TEXTLIST S3_Alarms
  0 = 'S3 0 Row 1 Failed To Advance.. Check Qxxx.x Default' | German: 'S3 0 Row 1 Failed To Advance.. Check Qxxx.x German' | French: 'S3 0 Row 1 Failed To Advance.. Check Qxxx.x French'
  1 = 'S3 1 Row 1 Failed To Return.. Check Qxxx.x Default' | German: 'S3 1 Row 1 Failed To Return.. Check Qxxx.x German' | French: 'S3 1 Row 1 Failed To Return.. Check Qxxx.x French'
  2 = 'S3 2 Row 1 Lost Advance Position... Check Ixxx.x Default' | German: 'S3 2 Row 1 Lost Advance Position... Check Ixxx.x German' | French: 'S3 2 Row 1 Lost Advance Position... Check Ixxx.x French'
  3 = 'S3 3 Row 1 Lost Return Position... Check Ixxx.x Default' | German: 'S3 3 Row 1 Lost Return Position... Check Ixxx.x German' | French: 'S3 3 Row 1 Lost Return Position... Check Ixxx.x French'
  4 = 'S3 4 Row 1 Switch Fault... Check Ixxx.x / Ixxx.x Default' | German: 'S3 4 Row 1 Switch Fault... Check Ixxx.x / Ixxx.x German' | French: 'S3 4 Row 1 Switch Fault... Check Ixxx.x / Ixxx.x French'
  5 = 'S3 5 Row 1 Spare Message Default' | German: 'S3 5 Row 1 Spare Message German' | French: 'S3 5 Row 1 Spare Message French'
  6 = 'S3 6 Row 1 Spare Message Default' | German: 'S3 6 Row 1 Spare Message German' | French: 'S3 6 Row 1 Spare Message French'
  7 = 'S3 7 Row 1 Spare Message Default' | German: 'S3 7 Row 1 Spare Message German' | French: 'S3 7 Row 1 Spare Message French'
  8 = 'S3 8 Row 1 Spare Message Default' | German: 'S3 8 Row 1 Spare Message German' | French: 'S3 8 Row 1 Spare Message French'
  9 = 'S3 9 Row 1 Spare Message Default' | German: 'S3 9 Row 1 Spare Message German' | French: 'S3 9 Row 1 Spare Message French'
  10 = 'S3 10 Row 2 Failed To Advance.. Check Qxxx.x Default' | German: 'S3 10 Row 2 Failed To Advance.. Check Qxxx.x German' | French: 'S3 10 Row 2 Failed To Advance.. Check Qxxx.x French'
  11 = 'S3 11 Row 2 Failed To Return.. Check Qxxx.x Default' | German: 'S3 11 Row 2 Failed To Return.. Check Qxxx.x German' | French: 'S3 11 Row 2 Failed To Return.. Check Qxxx.x French'
  12 = 'S3 12 Row 2 Lost Advance Position... Check Ixxx.x Default' | German: 'S3 12 Row 2 Lost Advance Position... Check Ixxx.x German' | French: 'S3 12 Row 2 Lost Advance Position... Check Ixxx.x French'
  13 = 'S3 13 Row 2 Lost Return Position... Check Ixxx.x Default' | German: 'S3 13 Row 2 Lost Return Position... Check Ixxx.x German' | French: 'S3 13 Row 2 Lost Return Position... Check Ixxx.x French'
  14 = 'S3 14 Row 2 Switch Fault... Check Ixxx.x / Ixxx.x Default' | German: 'S3 14 Row 2 Switch Fault... Check Ixxx.x / Ixxx.x German' | French: 'S3 14 Row 2 Switch Fault... Check Ixxx.x / Ixxx.x French'
  15 = 'S3 15 Row 2 Spare Message Default' | German: 'S3 15 Row 2 Spare Message German' | French: 'S3 15 Row 2 Spare Message French'
  16 = 'S3 16 Row 2 Spare Message Default' | German: 'S3 16 Row 2 Spare Message German' | French: 'S3 16 Row 2 Spare Message French'
  17 = 'S3 17 Row 2 Spare Message Default' | German: 'S3 17 Row 2 Spare Message German' | French: 'S3 17 Row 2 Spare Message French'
  18 = 'S3 18 Row 2 Spare Message Default' | German: 'S3 18 Row 2 Spare Message German' | French: 'S3 18 Row 2 Spare Message French'
  19 = 'S3 19 Row 2 Spare Message Default' | German: 'S3 19 Row 2 Spare Message German' | French: 'S3 19 Row 2 Spare Message French'
  20 = 'S3 20 Row 3 Failed To Advance.. Check Qxxx.x Default' | German: 'S3 20 Row 3 Failed To Advance.. Check Qxxx.x German' | French: 'S3 20 Row 3 Failed To Advance.. Check Qxxx.x French'
  21 = 'S3 21 Row 3 Failed To Return.. Check Qxxx.x Default' | German: 'S3 21 Row 3 Failed To Return.. Check Qxxx.x German' | French: 'S3 21 Row 3 Failed To Return.. Check Qxxx.x French'
  22 = 'S3 22 Row 3 Lost Advance Position... Check Ixxx.x Default' | German: 'S3 22 Row 3 Lost Advance Position... Check Ixxx.x German' | French: 'S3 22 Row 3 Lost Advance Position... Check Ixxx.x French'
  23 = 'S3 23 Row 3 Lost Return Position... Check Ixxx.x Default' | German: 'S3 23 Row 3 Lost Return Position... Check Ixxx.x German' | French: 'S3 23 Row 3 Lost Return Position... Check Ixxx.x French'
  24 = 'S3 24 Row 3 Switch Fault... Check Ixxx.x / Ixxx.x Default' | German: 'S3 24 Row 3 Switch Fault... Check Ixxx.x / Ixxx.x German' | French: 'S3 24 Row 3 Switch Fault... Check Ixxx.x / Ixxx.x French'
  25 = 'S3 25 Row 3 Spare Message Default' | German: 'S3 25 Row 3 Spare Message German' | French: 'S3 25 Row 3 Spare Message French'
  26 = 'S3 26 Row 3 Spare Message Default' | German: 'S3 26 Row 3 Spare Message German' | French: 'S3 26 Row 3 Spare Message French'
  27 = 'S3 27 Row 3 Spare Message Default' | German: 'S3 27 Row 3 Spare Message German' | French: 'S3 27 Row 3 Spare Message French'
  28 = 'S3 28 Row 3 Spare Message Default' | German: 'S3 28 Row 3 Spare Message German' | French: 'S3 28 Row 3 Spare Message French'
  29 = 'S3 29 Row 3 Spare Message Default' | German: 'S3 29 Row 3 Spare Message German' | French: 'S3 29 Row 3 Spare Message French'
  30 = 'S3 30 Row 4 Failed To Advance.. Check Qxxx.x Default' | German: 'S3 30 Row 4 Failed To Advance.. Check Qxxx.x German' | French: 'S3 30 Row 4 Failed To Advance.. Check Qxxx.x French'
  31 = 'S3 31 Row 4 Failed To Return.. Check Qxxx.x Default' | German: 'S3 31 Row 4 Failed To Return.. Check Qxxx.x German' | French: 'S3 31 Row 4 Failed To Return.. Check Qxxx.x French'
  32 = 'S3 32 Row 4 Lost Advance Position... Check Ixxx.x Default' | German: 'S3 32 Row 4 Lost Advance Position... Check Ixxx.x German' | French: 'S3 32 Row 4 Lost Advance Position... Check Ixxx.x French'
  33 = 'S3 33 Row 4 Lost Return Position... Check Ixxx.x Default' | German: 'S3 33 Row 4 Lost Return Position... Check Ixxx.x German' | French: 'S3 33 Row 4 Lost Return Position... Check Ixxx.x French'
  34 = 'S3 34 Row 4 Switch Fault... Check Ixxx.x / Ixxx.x Default' | German: 'S3 34 Row 4 Switch Fault... Check Ixxx.x / Ixxx.x German' | French: 'S3 34 Row 4 Switch Fault... Check Ixxx.x / Ixxx.x French'
  35 = 'S3 35 Row 4 Spare Message Default' | German: 'S3 35 Row 4 Spare Message German' | French: 'S3 35 Row 4 Spare Message French'
  36 = 'S3 36 Row 4 Spare Message Default' | German: 'S3 36 Row 4 Spare Message German' | French: 'S3 36 Row 4 Spare Message French'
  37 = 'S3 37 Row 4 Spare Message Default' | German: 'S3 37 Row 4 Spare Message German' | French: 'S3 37 Row 4 Spare Message French'
  38 = 'S3 38 Row 4 Spare Message Default' | German: 'S3 38 Row 4 Spare Message German' | French: 'S3 38 Row 4 Spare Message French'
  39 = 'S3 39 Row 4 Spare Message Default' | German: 'S3 39 Row 4 Spare Message German' | French: 'S3 39 Row 4 Spare Message French'
  40 = 'S3 40 Row 5 Failed To Advance.. Check Qxxx.x Default' | German: 'S3 40 Row 5 Failed To Advance.. Check Qxxx.x German' | French: 'S3 40 Row 5 Failed To Advance.. Check Qxxx.x French'
  41 = 'S3 41 Row 5 Failed To Return.. Check Qxxx.x Default' | German: 'S3 41 Row 5 Failed To Return.. Check Qxxx.x German' | French: 'S3 41 Row 5 Failed To Return.. Check Qxxx.x French'
  42 = 'S3 42 Row 5 Lost Advance Position... Check Ixxx.x Default' | German: 'S3 42 Row 5 Lost Advance Position... Check Ixxx.x German' | French: 'S3 42 Row 5 Lost Advance Position... Check Ixxx.x French'
  43 = 'S3 43 Row 5 Lost Return Position... Check Ixxx.x Default' | German: 'S3 43 Row 5 Lost Return Position... Check Ixxx.x German' | French: 'S3 43 Row 5 Lost Return Position... Check Ixxx.x French'
  44 = 'S3 44 Row 5 Switch Fault... Check Ixxx.x / Ixxx.x Default' | German: 'S3 44 Row 5 Switch Fault... Check Ixxx.x / Ixxx.x German' | French: 'S3 44 Row 5 Switch Fault... Check Ixxx.x / Ixxx.x French'
  45 = 'S3 45 Row 5 Spare Message Default' | German: 'S3 45 Row 5 Spare Message German' | French: 'S3 45 Row 5 Spare Message French'
  46 = 'S3 46 Row 5 Spare Message Default' | German: 'S3 46 Row 5 Spare Message German' | French: 'S3 46 Row 5 Spare Message French'
  47 = 'S3 47 Row 5 Spare Message Default' | German: 'S3 47 Row 5 Spare Message German' | French: 'S3 47 Row 5 Spare Message French'
  48 = 'S3 48 Row 5 Spare Message Default' | German: 'S3 48 Row 5 Spare Message German' | French: 'S3 48 Row 5 Spare Message French'
  49 = 'S3 49 Row 5 Spare Message Default' | German: 'S3 49 Row 5 Spare Message German' | French: 'S3 49 Row 5 Spare Message French'
  50 = 'S3 50 Row 6 Failed To Advance.. Check Qxxx.x Default' | German: 'S3 50 Row 6 Failed To Advance.. Check Qxxx.x German' | French: 'S3 50 Row 6 Failed To Advance.. Check Qxxx.x French'
  51 = 'S3 51 Row 6 Failed To Return.. Check Qxxx.x Default' | German: 'S3 51 Row 6 Failed To Return.. Check Qxxx.x German' | French: 'S3 51 Row 6 Failed To Return.. Check Qxxx.x French'
  52 = 'S3 52 Row 6 Lost Advance Position... Check Ixxx.x Default' | German: 'S3 52 Row 6 Lost Advance Position... Check Ixxx.x German' | French: 'S3 52 Row 6 Lost Advance Position... Check Ixxx.x French'
  53 = 'S3 53 Row 6 Lost Return Position... Check Ixxx.x Default' | German: 'S3 53 Row 6 Lost Return Position... Check Ixxx.x German' | French: 'S3 53 Row 6 Lost Return Position... Check Ixxx.x French'
  54 = 'S3 54 Row 6 Switch Fault... Check Ixxx.x / Ixxx.x Default' | German: 'S3 54 Row 6 Switch Fault... Check Ixxx.x / Ixxx.x German' | French: 'S3 54 Row 6 Switch Fault... Check Ixxx.x / Ixxx.x French'
  55 = 'S3 55 Row 6 Spare Message Default' | German: 'S3 55 Row 6 Spare Message German' | French: 'S3 55 Row 6 Spare Message French'
  56 = 'S3 56 Row 6 Spare Message Default' | German: 'S3 56 Row 6 Spare Message German' | French: 'S3 56 Row 6 Spare Message French'
  57 = 'S3 57 Row 6 Spare Message Default' | German: 'S3 57 Row 6 Spare Message German' | French: 'S3 57 Row 6 Spare Message French'
  58 = 'S3 58 Row 6 Spare Message Default' | German: 'S3 58 Row 6 Spare Message German' | French: 'S3 58 Row 6 Spare Message French'
  59 = 'S3 59 Row 6 Spare Message Default' | German: 'S3 59 Row 6 Spare Message German' | French: 'S3 59 Row 6 Spare Message French'
  60 = 'S3 60 Row 7 Failed To Advance.. Check Qxxx.x Default' | German: 'S3 60 Row 7 Failed To Advance.. Check Qxxx.x German' | French: 'S3 60 Row 7 Failed To Advance.. Check Qxxx.x French'
  61 = 'S3 61 Row 7 Failed To Return.. Check Qxxx.x Default' | German: 'S3 61 Row 7 Failed To Return.. Check Qxxx.x German' | French: 'S3 61 Row 7 Failed To Return.. Check Qxxx.x French'
  62 = 'S3 62 Row 7 Lost Advance Position... Check Ixxx.x Default' | German: 'S3 62 Row 7 Lost Advance Position... Check Ixxx.x German' | French: 'S3 62 Row 7 Lost Advance Position... Check Ixxx.x French'
  63 = 'S3 63 Row 7 Lost Return Position... Check Ixxx.x Default' | German: 'S3 63 Row 7 Lost Return Position... Check Ixxx.x German' | French: 'S3 63 Row 7 Lost Return Position... Check Ixxx.x French'
  64 = 'S3 64 Row 7 Switch Fault... Check Ixxx.x / Ixxx.x Default' | German: 'S3 64 Row 7 Switch Fault... Check Ixxx.x / Ixxx.x German' | French: 'S3 64 Row 7 Switch Fault... Check Ixxx.x / Ixxx.x French'
  65 = 'S3 65 Row 7 Spare Message Default' | German: 'S3 65 Row 7 Spare Message German' | French: 'S3 65 Row 7 Spare Message French'
  66 = 'S3 66 Row 7 Spare Message Default' | German: 'S3 66 Row 7 Spare Message German' | French: 'S3 66 Row 7 Spare Message French'
  67 = 'S3 67 Row 7 Spare Message Default' | German: 'S3 67 Row 7 Spare Message German' | French: 'S3 67 Row 7 Spare Message French'
  68 = 'S3 68 Row 7 Spare Message Default' | German: 'S3 68 Row 7 Spare Message German' | French: 'S3 68 Row 7 Spare Message French'
  69 = 'S3 69 Row 7 Spare Message Default' | German: 'S3 69 Row 7 Spare Message German' | French: 'S3 69 Row 7 Spare Message French'
  70 = 'S3 70 Row 8 Failed To Advance.. Check Qxxx.x Default' | German: 'S3 70 Row 8 Failed To Advance.. Check Qxxx.x German' | French: 'S3 70 Row 8 Failed To Advance.. Check Qxxx.x French'
  71 = 'S3 71 Row 8 Failed To Return.. Check Qxxx.x Default' | German: 'S3 71 Row 8 Failed To Return.. Check Qxxx.x German' | French: 'S3 71 Row 8 Failed To Return.. Check Qxxx.x French'
  72 = 'S3 72 Row 8 Lost Advance Position... Check Ixxx.x Default' | German: 'S3 72 Row 8 Lost Advance Position... Check Ixxx.x German' | French: 'S3 72 Row 8 Lost Advance Position... Check Ixxx.x French'
  73 = 'S3 73 Row 8 Lost Return Position... Check Ixxx.x Default' | German: 'S3 73 Row 8 Lost Return Position... Check Ixxx.x German' | French: 'S3 73 Row 8 Lost Return Position... Check Ixxx.x French'
  74 = 'S3 74 Row 8 Switch Fault... Check Ixxx.x / Ixxx.x Default' | German: 'S3 74 Row 8 Switch Fault... Check Ixxx.x / Ixxx.x German' | French: 'S3 74 Row 8 Switch Fault... Check Ixxx.x / Ixxx.x French'
  75 = 'S3 75 Row 8 Spare Message Default' | German: 'S3 75 Row 8 Spare Message German' | French: 'S3 75 Row 8 Spare Message French'
  76 = 'S3 76 Row 8 Spare Message Default' | German: 'S3 76 Row 8 Spare Message German' | French: 'S3 76 Row 8 Spare Message French'
  77 = 'S3 77 Row 8 Spare Message Default' | German: 'S3 77 Row 8 Spare Message German' | French: 'S3 77 Row 8 Spare Message French'
  78 = 'S3 78 Row 8 Spare Message Default' | German: 'S3 78 Row 8 Spare Message German' | French: 'S3 78 Row 8 Spare Message French'
  79 = 'S3 79 Row 8 Spare Message Default' | German: 'S3 79 Row 8 Spare Message German' | French: 'S3 79 Row 8 Spare Message French'
  80 = 'S3 80 Row 9 Failed To Advance.. Check Qxxx.x Default' | German: 'S3 80 Row 9 Failed To Advance.. Check Qxxx.x German' | French: 'S3 80 Row 9 Failed To Advance.. Check Qxxx.x French'
  81 = 'S3 81 Row 9 Failed To Return.. Check Qxxx.x Default' | German: 'S3 81 Row 9 Failed To Return.. Check Qxxx.x German' | French: 'S3 81 Row 9 Failed To Return.. Check Qxxx.x French'
  82 = 'S3 82 Row 9 Lost Advance Position... Check Ixxx.x Default' | German: 'S3 82 Row 9 Lost Advance Position... Check Ixxx.x German' | French: 'S3 82 Row 9 Lost Advance Position... Check Ixxx.x French'
  83 = 'S3 83 Row 9 Lost Return Position... Check Ixxx.x Default' | German: 'S3 83 Row 9 Lost Return Position... Check Ixxx.x German' | French: 'S3 83 Row 9 Lost Return Position... Check Ixxx.x French'
  84 = 'S3 84 Row 9 Switch Fault... Check Ixxx.x / Ixxx.x Default' | German: 'S3 84 Row 9 Switch Fault... Check Ixxx.x / Ixxx.x German' | French: 'S3 84 Row 9 Switch Fault... Check Ixxx.x / Ixxx.x French'
  85 = 'S3 85 Row 9 Spare Message Default' | German: 'S3 85 Row 9 Spare Message German' | French: 'S3 85 Row 9 Spare Message French'
  86 = 'S3 86 Row 9 Spare Message Default' | German: 'S3 86 Row 9 Spare Message German' | French: 'S3 86 Row 9 Spare Message French'
  87 = 'S3 87 Row 9 Spare Message Default' | German: 'S3 87 Row 9 Spare Message German' | French: 'S3 87 Row 9 Spare Message French'
  88 = 'S3 88 Row 9 Spare Message Default' | German: 'S3 88 Row 9 Spare Message German' | French: 'S3 88 Row 9 Spare Message French'
  89 = 'S3 89 Row 9 Spare Message Default' | German: 'S3 89 Row 9 Spare Message German' | French: 'S3 89 Row 9 Spare Message French'
  90 = 'S3 90 Row 10 Failed To Advance.. Check Qxxx.x Default' | German: 'S3 90 Row 10 Failed To Advance.. Check Qxxx.x German' | French: 'S3 90 Row 10 Failed To Advance.. Check Qxxx.x French'
  91 = 'S3 91 Row 10 Failed To Return.. Check Qxxx.x Default' | German: 'S3 91 Row 10 Failed To Return.. Check Qxxx.x German' | French: 'S3 91 Row 10 Failed To Return.. Check Qxxx.x French'
  92 = 'S3 92 Row 10 Lost Advance Position... Check Ixxx.x Default' | German: 'S3 92 Row 10 Lost Advance Position... Check Ixxx.x German' | French: 'S3 92 Row 10 Lost Advance Position... Check Ixxx.x French'
  93 = 'S3 93 Row 10 Lost Return Position... Check Ixxx.x Default' | German: 'S3 93 Row 10 Lost Return Position... Check Ixxx.x German' | French: 'S3 93 Row 10 Lost Return Position... Check Ixxx.x French'
  94 = 'S3 94 Row 10 Switch Fault... Check Ixxx.x / Ixxx.x Default' | German: 'S3 94 Row 10 Switch Fault... Check Ixxx.x / Ixxx.x German' | French: 'S3 94 Row 10 Switch Fault... Check Ixxx.x / Ixxx.x French'
  95 = 'S3 95 Row 10 Spare Message Default' | German: 'S3 95 Row 10 Spare Message German' | French: 'S3 95 Row 10 Spare Message French'
  96 = 'S3 96 Row 10 Spare Message Default' | German: 'S3 96 Row 10 Spare Message German' | French: 'S3 96 Row 10 Spare Message French'
  97 = 'S3 97 Row 10 Spare Message Default' | German: 'S3 97 Row 10 Spare Message German' | French: 'S3 97 Row 10 Spare Message French'
  98 = 'S3 98 Row 10 Spare Message Default' | German: 'S3 98 Row 10 Spare Message German' | French: 'S3 98 Row 10 Spare Message French'
  99 = 'S3 99 Row 10 Spare Message Default' | German: 'S3 99 Row 10 Spare Message German' | French: 'S3 99 Row 10 Spare Message French'
  100 = 'S3 100 Row 11 Failed To Advance.. Check Qxxx.x Default' | German: 'S3 100 Row 11 Failed To Advance.. Check Qxxx.x German' | French: 'S3 100 Row 11 Failed To Advance.. Check Qxxx.x French'
  101 = 'S3 101 Row 11 Failed To Return.. Check Qxxx.x Default' | German: 'S3 101 Row 11 Failed To Return.. Check Qxxx.x German' | French: 'S3 101 Row 11 Failed To Return.. Check Qxxx.x French'
  102 = 'S3 102 Row 11 Lost Advance Position... Check Ixxx.x Default' | German: 'S3 102 Row 11 Lost Advance Position... Check Ixxx.x German' | French: 'S3 102 Row 11 Lost Advance Position... Check Ixxx.x French'
  103 = 'S3 103 Row 11 Lost Return Position... Check Ixxx.x Default' | German: 'S3 103 Row 11 Lost Return Position... Check Ixxx.x German' | French: 'S3 103 Row 11 Lost Return Position... Check Ixxx.x French'
  104 = 'S3 104 Row 11 Switch Fault... Check Ixxx.x / Ixxx.x Default' | German: 'S3 104 Row 11 Switch Fault... Check Ixxx.x / Ixxx.x German' | French: 'S3 104 Row 11 Switch Fault... Check Ixxx.x / Ixxx.x French'
  105 = 'S3 105 Row 11 Spare Message Default' | German: 'S3 105 Row 11 Spare Message German' | French: 'S3 105 Row 11 Spare Message French'
  106 = 'S3 106 Row 11 Spare Message Default' | German: 'S3 106 Row 11 Spare Message German' | French: 'S3 106 Row 11 Spare Message French'
  107 = 'S3 107 Row 11 Spare Message Default' | German: 'S3 107 Row 11 Spare Message German' | French: 'S3 107 Row 11 Spare Message French'
  108 = 'S3 108 Row 11 Spare Message Default' | German: 'S3 108 Row 11 Spare Message German' | French: 'S3 108 Row 11 Spare Message French'
  109 = 'S3 109 Row 11 Spare Message Default' | German: 'S3 109 Row 11 Spare Message German' | French: 'S3 109 Row 11 Spare Message French'
  110 = 'S3 110 Row 12 Failed To Advance.. Check Qxxx.x Default' | German: 'S3 110 Row 12 Failed To Advance.. Check Qxxx.x German' | French: 'S3 110 Row 12 Failed To Advance.. Check Qxxx.x French'
  111 = 'S3 111 Row 12 Failed To Return.. Check Qxxx.x Default' | German: 'S3 111 Row 12 Failed To Return.. Check Qxxx.x German' | French: 'S3 111 Row 12 Failed To Return.. Check Qxxx.x French'
  112 = 'S3 112 Row 12 Lost Advance Position... Check Ixxx.x Default' | German: 'S3 112 Row 12 Lost Advance Position... Check Ixxx.x German' | French: 'S3 112 Row 12 Lost Advance Position... Check Ixxx.x French'
  113 = 'S3 113 Row 12 Lost Return Position... Check Ixxx.x Default' | German: 'S3 113 Row 12 Lost Return Position... Check Ixxx.x German' | French: 'S3 113 Row 12 Lost Return Position... Check Ixxx.x French'
  114 = 'S3 114 Row 12 Switch Fault... Check Ixxx.x / Ixxx.x Default' | German: 'S3 114 Row 12 Switch Fault... Check Ixxx.x / Ixxx.x German' | French: 'S3 114 Row 12 Switch Fault... Check Ixxx.x / Ixxx.x French'
  115 = 'S3 115 Row 12 Spare Message Default' | German: 'S3 115 Row 12 Spare Message German' | French: 'S3 115 Row 12 Spare Message French'
  116 = 'S3 116 Row 12 Spare Message Default' | German: 'S3 116 Row 12 Spare Message German' | French: 'S3 116 Row 12 Spare Message French'
  117 = 'S3 117 Row 12 Spare Message Default' | German: 'S3 117 Row 12 Spare Message German' | French: 'S3 117 Row 12 Spare Message French'
  118 = 'S3 118 Row 12 Spare Message Default' | German: 'S3 118 Row 12 Spare Message German' | French: 'S3 118 Row 12 Spare Message French'
  119 = 'S3 119 Row 12 Spare Message Default' | German: 'S3 119 Row 12 Spare Message German' | French: 'S3 119 Row 12 Spare Message French'
  120 = 'S3 120 Row 13 Failed To Advance.. Check Qxxx.x Default' | German: 'S3 120 Row 13 Failed To Advance.. Check Qxxx.x German' | French: 'S3 120 Row 13 Failed To Advance.. Check Qxxx.x French'
  121 = 'S3 121 Row 13 Failed To Return.. Check Qxxx.x Default' | German: 'S3 121 Row 13 Failed To Return.. Check Qxxx.x German' | French: 'S3 121 Row 13 Failed To Return.. Check Qxxx.x French'
  122 = 'S3 122 Row 13 Lost Advance Position... Check Ixxx.x Default' | German: 'S3 122 Row 13 Lost Advance Position... Check Ixxx.x German' | French: 'S3 122 Row 13 Lost Advance Position... Check Ixxx.x French'
  123 = 'S3 123 Row 13 Lost Return Position... Check Ixxx.x Default' | German: 'S3 123 Row 13 Lost Return Position... Check Ixxx.x German' | French: 'S3 123 Row 13 Lost Return Position... Check Ixxx.x French'
  124 = 'S3 124 Row 13 Switch Fault... Check Ixxx.x / Ixxx.x Default' | German: 'S3 124 Row 13 Switch Fault... Check Ixxx.x / Ixxx.x German' | French: 'S3 124 Row 13 Switch Fault... Check Ixxx.x / Ixxx.x French'
  125 = 'S3 125 Row 13 Spare Message Default' | German: 'S3 125 Row 13 Spare Message German' | French: 'S3 125 Row 13 Spare Message French'
  126 = 'S3 126 Row 13 Spare Message Default' | German: 'S3 126 Row 13 Spare Message German' | French: 'S3 126 Row 13 Spare Message French'
  127 = 'S3 127 Row 13 Spare Message Default' | German: 'S3 127 Row 13 Spare Message German' | French: 'S3 127 Row 13 Spare Message French'
  128 = 'S3 128 Row 13 Spare Message Default' | German: 'S3 128 Row 13 Spare Message German' | French: 'S3 128 Row 13 Spare Message French'
  129 = 'S3 129 Row 13 Spare Message Default' | German: 'S3 129 Row 13 Spare Message German' | French: 'S3 129 Row 13 Spare Message French'
  130 = 'S3 130 Row 14 Failed To Advance.. Check Qxxx.x Default' | German: 'S3 130 Row 14 Failed To Advance.. Check Qxxx.x German' | French: 'S3 130 Row 14 Failed To Advance.. Check Qxxx.x French'
  131 = 'S3 131 Row 14 Failed To Return.. Check Qxxx.x Default' | German: 'S3 131 Row 14 Failed To Return.. Check Qxxx.x German' | French: 'S3 131 Row 14 Failed To Return.. Check Qxxx.x French'
  132 = 'S3 132 Row 14 Lost Advance Position... Check Ixxx.x Default' | German: 'S3 132 Row 14 Lost Advance Position... Check Ixxx.x German' | French: 'S3 132 Row 14 Lost Advance Position... Check Ixxx.x French'
  133 = 'S3 133 Row 14 Lost Return Position... Check Ixxx.x Default' | German: 'S3 133 Row 14 Lost Return Position... Check Ixxx.x German' | French: 'S3 133 Row 14 Lost Return Position... Check Ixxx.x French'
  134 = 'S3 134 Row 14 Switch Fault... Check Ixxx.x / Ixxx.x Default' | German: 'S3 134 Row 14 Switch Fault... Check Ixxx.x / Ixxx.x German' | French: 'S3 134 Row 14 Switch Fault... Check Ixxx.x / Ixxx.x French'
  135 = 'S3 135 Row 14 Spare Message Default' | German: 'S3 135 Row 14 Spare Message German' | French: 'S3 135 Row 14 Spare Message French'
  136 = 'S3 136 Row 14 Spare Message Default' | German: 'S3 136 Row 14 Spare Message German' | French: 'S3 136 Row 14 Spare Message French'
  137 = 'S3 137 Row 14 Spare Message Default' | German: 'S3 137 Row 14 Spare Message German' | French: 'S3 137 Row 14 Spare Message French'
  138 = 'S3 138 Row 14 Spare Message Default' | German: 'S3 138 Row 14 Spare Message German' | French: 'S3 138 Row 14 Spare Message French'
  139 = 'S3 139 Row 14 Spare Message Default' | German: 'S3 139 Row 14 Spare Message German' | French: 'S3 139 Row 14 Spare Message French'
  140 = 'S3 140 Row 15 Failed To Advance.. Check Qxxx.x Default' | German: 'S3 140 Row 15 Failed To Advance.. Check Qxxx.x German' | French: 'S3 140 Row 15 Failed To Advance.. Check Qxxx.x French'
  141 = 'S3 141 Row 15 Failed To Return.. Check Qxxx.x Default' | German: 'S3 141 Row 15 Failed To Return.. Check Qxxx.x German' | French: 'S3 141 Row 15 Failed To Return.. Check Qxxx.x French'
  142 = 'S3 142 Row 15 Lost Advance Position... Check Ixxx.x Default' | German: 'S3 142 Row 15 Lost Advance Position... Check Ixxx.x German' | French: 'S3 142 Row 15 Lost Advance Position... Check Ixxx.x French'
  143 = 'S3 143 Row 15 Lost Return Position... Check Ixxx.x Default' | German: 'S3 143 Row 15 Lost Return Position... Check Ixxx.x German' | French: 'S3 143 Row 15 Lost Return Position... Check Ixxx.x French'
  144 = 'S3 144 Row 15 Switch Fault... Check Ixxx.x / Ixxx.x Default' | German: 'S3 144 Row 15 Switch Fault... Check Ixxx.x / Ixxx.x German' | French: 'S3 144 Row 15 Switch Fault... Check Ixxx.x / Ixxx.x French'
  145 = 'S3 145 Row 15 Spare Message Default' | German: 'S3 145 Row 15 Spare Message German' | French: 'S3 145 Row 15 Spare Message French'
  146 = 'S3 146 Row 15 Spare Message Default' | German: 'S3 146 Row 15 Spare Message German' | French: 'S3 146 Row 15 Spare Message French'
  147 = 'S3 147 Row 15 Spare Message Default' | German: 'S3 147 Row 15 Spare Message German' | French: 'S3 147 Row 15 Spare Message French'
  148 = 'S3 148 Row 15 Spare Message Default' | German: 'S3 148 Row 15 Spare Message German' | French: 'S3 148 Row 15 Spare Message French'
  149 = 'S3 149 Row 15 Spare Message Default' | German: 'S3 149 Row 15 Spare Message German' | French: 'S3 149 Row 15 Spare Message French'
  150 = 'S3 150 Row 16 Failed To Advance.. Check Qxxx.x Default' | German: 'S3 150 Row 16 Failed To Advance.. Check Qxxx.x German' | French: 'S3 150 Row 16 Failed To Advance.. Check Qxxx.x French'
  151 = 'S3 151 Row 16 Failed To Return.. Check Qxxx.x Default' | German: 'S3 151 Row 16 Failed To Return.. Check Qxxx.x German' | French: 'S3 151 Row 16 Failed To Return.. Check Qxxx.x French'
  152 = 'S3 152 Row 16 Lost Advance Position... Check Ixxx.x Default' | German: 'S3 152 Row 16 Lost Advance Position... Check Ixxx.x German' | French: 'S3 152 Row 16 Lost Advance Position... Check Ixxx.x French'
  153 = 'S3 153 Row 16 Lost Return Position... Check Ixxx.x Default' | German: 'S3 153 Row 16 Lost Return Position... Check Ixxx.x German' | French: 'S3 153 Row 16 Lost Return Position... Check Ixxx.x French'
  154 = 'S3 154 Row 16 Switch Fault... Check Ixxx.x / Ixxx.x Default' | German: 'S3 154 Row 16 Switch Fault... Check Ixxx.x / Ixxx.x German' | French: 'S3 154 Row 16 Switch Fault... Check Ixxx.x / Ixxx.x French'
  155 = 'S3 155 Row 16 Spare Message Default' | German: 'S3 155 Row 16 Spare Message German' | French: 'S3 155 Row 16 Spare Message French'
  156 = 'S3 156 Row 16 Spare Message Default' | German: 'S3 156 Row 16 Spare Message German' | French: 'S3 156 Row 16 Spare Message French'
  157 = 'S3 157 Row 16 Spare Message Default' | German: 'S3 157 Row 16 Spare Message German' | French: 'S3 157 Row 16 Spare Message French'
  158 = 'S3 158 Row 16 Spare Message Default' | German: 'S3 158 Row 16 Spare Message German' | French: 'S3 158 Row 16 Spare Message French'
  159 = 'S3 159 Row 16 Spare Message Default' | German: 'S3 159 Row 16 Spare Message German' | French: 'S3 159 Row 16 Spare Message French'
  160 = 'S3 160 Row 17 Failed To Advance.. Check Qxxx.x Default' | German: 'S3 160 Row 17 Failed To Advance.. Check Qxxx.x German' | French: 'S3 160 Row 17 Failed To Advance.. Check Qxxx.x French'
  161 = 'S3 161 Row 17 Failed To Return.. Check Qxxx.x Default' | German: 'S3 161 Row 17 Failed To Return.. Check Qxxx.x German' | French: 'S3 161 Row 17 Failed To Return.. Check Qxxx.x French'
  162 = 'S3 162 Row 17 Lost Advance Position... Check Ixxx.x Default' | German: 'S3 162 Row 17 Lost Advance Position... Check Ixxx.x German' | French: 'S3 162 Row 17 Lost Advance Position... Check Ixxx.x French'
  163 = 'S3 163 Row 17 Lost Return Position... Check Ixxx.x Default' | German: 'S3 163 Row 17 Lost Return Position... Check Ixxx.x German' | French: 'S3 163 Row 17 Lost Return Position... Check Ixxx.x French'
  164 = 'S3 164 Row 17 Switch Fault... Check Ixxx.x / Ixxx.x Default' | German: 'S3 164 Row 17 Switch Fault... Check Ixxx.x / Ixxx.x German' | French: 'S3 164 Row 17 Switch Fault... Check Ixxx.x / Ixxx.x French'
  165 = 'S3 165 Row 17 Spare Message Default' | German: 'S3 165 Row 17 Spare Message German' | French: 'S3 165 Row 17 Spare Message French'
  166 = 'S3 166 Row 17 Spare Message Default' | German: 'S3 166 Row 17 Spare Message German' | French: 'S3 166 Row 17 Spare Message French'
  167 = 'S3 167 Row 17 Spare Message Default' | German: 'S3 167 Row 17 Spare Message German' | French: 'S3 167 Row 17 Spare Message French'
  168 = 'S3 168 Row 17 Spare Message Default' | German: 'S3 168 Row 17 Spare Message German' | French: 'S3 168 Row 17 Spare Message French'
  169 = 'S3 169 Row 17 Spare Message Default' | German: 'S3 169 Row 17 Spare Message German' | French: 'S3 169 Row 17 Spare Message French'
  170 = 'S3 170 Row 18 Failed To Advance.. Check Qxxx.x Default' | German: 'S3 170 Row 18 Failed To Advance.. Check Qxxx.x German' | French: 'S3 170 Row 18 Failed To Advance.. Check Qxxx.x French'
  171 = 'S3 171 Row 18 Failed To Return.. Check Qxxx.x Default' | German: 'S3 171 Row 18 Failed To Return.. Check Qxxx.x German' | French: 'S3 171 Row 18 Failed To Return.. Check Qxxx.x French'
  172 = 'S3 172 Row 18 Lost Advance Position... Check Ixxx.x Default' | German: 'S3 172 Row 18 Lost Advance Position... Check Ixxx.x German' | French: 'S3 172 Row 18 Lost Advance Position... Check Ixxx.x French'
  173 = 'S3 173 Row 18 Lost Return Position... Check Ixxx.x Default' | German: 'S3 173 Row 18 Lost Return Position... Check Ixxx.x German' | French: 'S3 173 Row 18 Lost Return Position... Check Ixxx.x French'
  174 = 'S3 174 Row 18 Switch Fault... Check Ixxx.x / Ixxx.x Default' | German: 'S3 174 Row 18 Switch Fault... Check Ixxx.x / Ixxx.x German' | French: 'S3 174 Row 18 Switch Fault... Check Ixxx.x / Ixxx.x French'
  175 = 'S3 175 Row 18 Spare Message Default' | German: 'S3 175 Row 18 Spare Message German' | French: 'S3 175 Row 18 Spare Message French'
  176 = 'S3 176 Row 18 Spare Message Default' | German: 'S3 176 Row 18 Spare Message German' | French: 'S3 176 Row 18 Spare Message French'
  177 = 'S3 177 Row 18 Spare Message Default' | German: 'S3 177 Row 18 Spare Message German' | French: 'S3 177 Row 18 Spare Message French'
  178 = 'S3 178 Row 18 Spare Message Default' | German: 'S3 178 Row 18 Spare Message German' | French: 'S3 178 Row 18 Spare Message French'
  179 = 'S3 179 Row 18 Spare Message Default' | German: 'S3 179 Row 18 Spare Message German' | French: 'S3 179 Row 18 Spare Message French'
  180 = 'S3 180 Row 19 Failed To Advance.. Check Qxxx.x Default' | German: 'S3 180 Row 19 Failed To Advance.. Check Qxxx.x German' | French: 'S3 180 Row 19 Failed To Advance.. Check Qxxx.x French'
  181 = 'S3 181 Row 19 Failed To Return.. Check Qxxx.x Default' | German: 'S3 181 Row 19 Failed To Return.. Check Qxxx.x German' | French: 'S3 181 Row 19 Failed To Return.. Check Qxxx.x French'
  182 = 'S3 182 Row 19 Lost Advance Position... Check Ixxx.x Default' | German: 'S3 182 Row 19 Lost Advance Position... Check Ixxx.x German' | French: 'S3 182 Row 19 Lost Advance Position... Check Ixxx.x French'
  183 = 'S3 183 Row 19 Lost Return Position... Check Ixxx.x Default' | German: 'S3 183 Row 19 Lost Return Position... Check Ixxx.x German' | French: 'S3 183 Row 19 Lost Return Position... Check Ixxx.x French'
  184 = 'S3 184 Row 19 Switch Fault... Check Ixxx.x / Ixxx.x Default' | German: 'S3 184 Row 19 Switch Fault... Check Ixxx.x / Ixxx.x German' | French: 'S3 184 Row 19 Switch Fault... Check Ixxx.x / Ixxx.x French'
  185 = 'S3 185 Row 19 Spare Message Default' | German: 'S3 185 Row 19 Spare Message German' | French: 'S3 185 Row 19 Spare Message French'
  186 = 'S3 186 Row 19 Spare Message Default' | German: 'S3 186 Row 19 Spare Message German' | French: 'S3 186 Row 19 Spare Message French'
  187 = 'S3 187 Row 19 Spare Message Default' | German: 'S3 187 Row 19 Spare Message German' | French: 'S3 187 Row 19 Spare Message French'
  188 = 'S3 188 Row 19 Spare Message Default' | German: 'S3 188 Row 19 Spare Message German' | French: 'S3 188 Row 19 Spare Message French'
  189 = 'S3 189 Row 19 Spare Message Default' | German: 'S3 189 Row 19 Spare Message German' | French: 'S3 189 Row 19 Spare Message French'
  190 = 'S3 190 Row 20 Failed To Advance.. Check Qxxx.x Default' | German: 'S3 190 Row 20 Failed To Advance.. Check Qxxx.x German' | French: 'S3 190 Row 20 Failed To Advance.. Check Qxxx.x French'
  191 = 'S3 191 Row 20 Failed To Return.. Check Qxxx.x Default' | German: 'S3 191 Row 20 Failed To Return.. Check Qxxx.x German' | French: 'S3 191 Row 20 Failed To Return.. Check Qxxx.x French'
  192 = 'S3 192 Row 20 Lost Advance Position... Check Ixxx.x Default' | German: 'S3 192 Row 20 Lost Advance Position... Check Ixxx.x German' | French: 'S3 192 Row 20 Lost Advance Position... Check Ixxx.x French'
  193 = 'S3 193 Row 20 Lost Return Position... Check Ixxx.x Default' | German: 'S3 193 Row 20 Lost Return Position... Check Ixxx.x German' | French: 'S3 193 Row 20 Lost Return Position... Check Ixxx.x French'
  194 = 'S3 194 Row 20 Switch Fault... Check Ixxx.x / Ixxx.x Default' | German: 'S3 194 Row 20 Switch Fault... Check Ixxx.x / Ixxx.x German' | French: 'S3 194 Row 20 Switch Fault... Check Ixxx.x / Ixxx.x French'
  195 = 'S3 195 Row 20 Spare Message Default' | German: 'S3 195 Row 20 Spare Message German' | French: 'S3 195 Row 20 Spare Message French'
  196 = 'S3 196 Row 20 Spare Message Default' | German: 'S3 196 Row 20 Spare Message German' | French: 'S3 196 Row 20 Spare Message French'
  197 = 'S3 197 Row 20 Spare Message Default' | German: 'S3 197 Row 20 Spare Message German' | French: 'S3 197 Row 20 Spare Message French'
  198 = 'S3 198 Row 20 Spare Message Default' | German: 'S3 198 Row 20 Spare Message German' | French: 'S3 198 Row 20 Spare Message French'
  199 = 'S3 199 Row 20 Spare Message Default' | German: 'S3 199 Row 20 Spare Message German' | French: 'S3 199 Row 20 Spare Message French'
  200 = 'S3 200 Row 21 Failed To Advance.. Check Qxxx.x Default' | German: 'S3 200 Row 21 Failed To Advance.. Check Qxxx.x German' | French: 'S3 200 Row 21 Failed To Advance.. Check Qxxx.x French'
  201 = 'S3 201 Row 21 Failed To Return.. Check Qxxx.x Default' | German: 'S3 201 Row 21 Failed To Return.. Check Qxxx.x German' | French: 'S3 201 Row 21 Failed To Return.. Check Qxxx.x French'
  202 = 'S3 202 Row 21 Lost Advance Position... Check Ixxx.x Default' | German: 'S3 202 Row 21 Lost Advance Position... Check Ixxx.x German' | French: 'S3 202 Row 21 Lost Advance Position... Check Ixxx.x French'
  203 = 'S3 203 Row 21 Lost Return Position... Check Ixxx.x Default' | German: 'S3 203 Row 21 Lost Return Position... Check Ixxx.x German' | French: 'S3 203 Row 21 Lost Return Position... Check Ixxx.x French'
  204 = 'S3 204 Row 21 Switch Fault... Check Ixxx.x / Ixxx.x Default' | German: 'S3 204 Row 21 Switch Fault... Check Ixxx.x / Ixxx.x German' | French: 'S3 204 Row 21 Switch Fault... Check Ixxx.x / Ixxx.x French'
  205 = 'S3 205 Row 21 Spare Message Default' | German: 'S3 205 Row 21 Spare Message German' | French: 'S3 205 Row 21 Spare Message French'
  206 = 'S3 206 Row 21 Spare Message Default' | German: 'S3 206 Row 21 Spare Message German' | French: 'S3 206 Row 21 Spare Message French'
  207 = 'S3 207 Row 21 Spare Message Default' | German: 'S3 207 Row 21 Spare Message German' | French: 'S3 207 Row 21 Spare Message French'
  208 = 'S3 208 Row 21 Spare Message Default' | German: 'S3 208 Row 21 Spare Message German' | French: 'S3 208 Row 21 Spare Message French'
  209 = 'S3 209 Row 21 Spare Message Default' | German: 'S3 209 Row 21 Spare Message German' | French: 'S3 209 Row 21 Spare Message French'
  210 = 'S3 210 Row 22 Failed To Advance.. Check Qxxx.x Default' | German: 'S3 210 Row 22 Failed To Advance.. Check Qxxx.x German' | French: 'S3 210 Row 22 Failed To Advance.. Check Qxxx.x French'
  211 = 'S3 211 Row 22 Failed To Return.. Check Qxxx.x Default' | German: 'S3 211 Row 22 Failed To Return.. Check Qxxx.x German' | French: 'S3 211 Row 22 Failed To Return.. Check Qxxx.x French'
  212 = 'S3 212 Row 22 Lost Advance Position... Check Ixxx.x Default' | German: 'S3 212 Row 22 Lost Advance Position... Check Ixxx.x German' | French: 'S3 212 Row 22 Lost Advance Position... Check Ixxx.x French'
  213 = 'S3 213 Row 22 Lost Return Position... Check Ixxx.x Default' | German: 'S3 213 Row 22 Lost Return Position... Check Ixxx.x German' | French: 'S3 213 Row 22 Lost Return Position... Check Ixxx.x French'
  214 = 'S3 214 Row 22 Switch Fault... Check Ixxx.x / Ixxx.x Default' | German: 'S3 214 Row 22 Switch Fault... Check Ixxx.x / Ixxx.x German' | French: 'S3 214 Row 22 Switch Fault... Check Ixxx.x / Ixxx.x French'
  215 = 'S3 215 Row 22 Spare Message Default' | German: 'S3 215 Row 22 Spare Message German' | French: 'S3 215 Row 22 Spare Message French'
  216 = 'S3 216 Row 22 Spare Message Default' | German: 'S3 216 Row 22 Spare Message German' | French: 'S3 216 Row 22 Spare Message French'
  217 = 'S3 217 Row 22 Spare Message Default' | German: 'S3 217 Row 22 Spare Message German' | French: 'S3 217 Row 22 Spare Message French'
  218 = 'S3 218 Row 22 Spare Message Default' | German: 'S3 218 Row 22 Spare Message German' | French: 'S3 218 Row 22 Spare Message French'
  219 = 'S3 219 Row 22 Spare Message Default' | German: 'S3 219 Row 22 Spare Message German' | French: 'S3 219 Row 22 Spare Message French'
  220 = 'S3 220 Row 23 Failed To Advance.. Check Qxxx.x Default' | German: 'S3 220 Row 23 Failed To Advance.. Check Qxxx.x German' | French: 'S3 220 Row 23 Failed To Advance.. Check Qxxx.x French'
  221 = 'S3 221 Row 23 Failed To Return.. Check Qxxx.x Default' | German: 'S3 221 Row 23 Failed To Return.. Check Qxxx.x German' | French: 'S3 221 Row 23 Failed To Return.. Check Qxxx.x French'
  222 = 'S3 222 Row 23 Lost Advance Position... Check Ixxx.x Default' | German: 'S3 222 Row 23 Lost Advance Position... Check Ixxx.x German' | French: 'S3 222 Row 23 Lost Advance Position... Check Ixxx.x French'
  223 = 'S3 223 Row 23 Lost Return Position... Check Ixxx.x Default' | German: 'S3 223 Row 23 Lost Return Position... Check Ixxx.x German' | French: 'S3 223 Row 23 Lost Return Position... Check Ixxx.x French'
  224 = 'S3 224 Row 23 Switch Fault... Check Ixxx.x / Ixxx.x Default' | German: 'S3 224 Row 23 Switch Fault... Check Ixxx.x / Ixxx.x German' | French: 'S3 224 Row 23 Switch Fault... Check Ixxx.x / Ixxx.x French'
  225 = 'S3 225 Row 23 Spare Message Default' | German: 'S3 225 Row 23 Spare Message German' | French: 'S3 225 Row 23 Spare Message French'
  226 = 'S3 226 Row 23 Spare Message Default' | German: 'S3 226 Row 23 Spare Message German' | French: 'S3 226 Row 23 Spare Message French'
  227 = 'S3 227 Row 23 Spare Message Default' | German: 'S3 227 Row 23 Spare Message German' | French: 'S3 227 Row 23 Spare Message French'
  228 = 'S3 228 Row 23 Spare Message Default' | German: 'S3 228 Row 23 Spare Message German' | French: 'S3 228 Row 23 Spare Message French'
  229 = 'S3 229 Row 23 Spare Message Default' | German: 'S3 229 Row 23 Spare Message German' | French: 'S3 229 Row 23 Spare Message French'
  230 = 'S3 230 Row 24 Failed To Advance.. Check Qxxx.x Default' | German: 'S3 230 Row 24 Failed To Advance.. Check Qxxx.x German' | French: 'S3 230 Row 24 Failed To Advance.. Check Qxxx.x French'
  231 = 'S3 231 Row 24 Failed To Return.. Check Qxxx.x Default' | German: 'S3 231 Row 24 Failed To Return.. Check Qxxx.x German' | French: 'S3 231 Row 24 Failed To Return.. Check Qxxx.x French'
  232 = 'S3 232 Row 24 Lost Advance Position... Check Ixxx.x Default' | German: 'S3 232 Row 24 Lost Advance Position... Check Ixxx.x German' | French: 'S3 232 Row 24 Lost Advance Position... Check Ixxx.x French'
  233 = 'S3 233 Row 24 Lost Return Position... Check Ixxx.x Default' | German: 'S3 233 Row 24 Lost Return Position... Check Ixxx.x German' | French: 'S3 233 Row 24 Lost Return Position... Check Ixxx.x French'
  234 = 'S3 234 Row 24 Switch Fault... Check Ixxx.x / Ixxx.x Default' | German: 'S3 234 Row 24 Switch Fault... Check Ixxx.x / Ixxx.x German' | French: 'S3 234 Row 24 Switch Fault... Check Ixxx.x / Ixxx.x French'
  235 = 'S3 235 Row 24 Spare Message Default' | German: 'S3 235 Row 24 Spare Message German' | French: 'S3 235 Row 24 Spare Message French'
  236 = 'S3 236 Row 24 Spare Message Default' | German: 'S3 236 Row 24 Spare Message German' | French: 'S3 236 Row 24 Spare Message French'
  237 = 'S3 237 Row 24 Spare Message Default' | German: 'S3 237 Row 24 Spare Message German' | French: 'S3 237 Row 24 Spare Message French'
  238 = 'S3 238 Row 24 Spare Message Default' | German: 'S3 238 Row 24 Spare Message German' | French: 'S3 238 Row 24 Spare Message French'
  239 = 'S3 239 Row 24 Spare Message Default' | German: 'S3 239 Row 24 Spare Message German' | French: 'S3 239 Row 24 Spare Message French'
  240 = 'S3 240 Row 25 Failed To Advance.. Check Qxxx.x Default' | German: 'S3 240 Row 25 Failed To Advance.. Check Qxxx.x German' | French: 'S3 240 Row 25 Failed To Advance.. Check Qxxx.x French'
  241 = 'S3 241 Row 25 Failed To Return.. Check Qxxx.x Default' | German: 'S3 241 Row 25 Failed To Return.. Check Qxxx.x German' | French: 'S3 241 Row 25 Failed To Return.. Check Qxxx.x French'
  242 = 'S3 242 Row 25 Lost Advance Position... Check Ixxx.x Default' | German: 'S3 242 Row 25 Lost Advance Position... Check Ixxx.x German' | French: 'S3 242 Row 25 Lost Advance Position... Check Ixxx.x French'
  243 = 'S3 243 Row 25 Lost Return Position... Check Ixxx.x Default' | German: 'S3 243 Row 25 Lost Return Position... Check Ixxx.x German' | French: 'S3 243 Row 25 Lost Return Position... Check Ixxx.x French'
  244 = 'S3 244 Row 25 Switch Fault... Check Ixxx.x / Ixxx.x Default' | German: 'S3 244 Row 25 Switch Fault... Check Ixxx.x / Ixxx.x German' | French: 'S3 244 Row 25 Switch Fault... Check Ixxx.x / Ixxx.x French'
  245 = 'S3 245 Row 25 Spare Message Default' | German: 'S3 245 Row 25 Spare Message German' | French: 'S3 245 Row 25 Spare Message French'
  246 = 'S3 246 Row 25 Spare Message Default' | German: 'S3 246 Row 25 Spare Message German' | French: 'S3 246 Row 25 Spare Message French'
  247 = 'S3 247 Row 25 Spare Message Default' | German: 'S3 247 Row 25 Spare Message German' | French: 'S3 247 Row 25 Spare Message French'
  248 = 'S3 248 Row 25 Spare Message Default' | German: 'S3 248 Row 25 Spare Message German' | French: 'S3 248 Row 25 Spare Message French'
  249 = 'S3 249 Row 25 Spare Message Default' | German: 'S3 249 Row 25 Spare Message German' | French: 'S3 249 Row 25 Spare Message French'
  250 = 'S3 250 Row 26 Failed To Advance.. Check Qxxx.x Default' | German: 'S3 250 Row 26 Failed To Advance.. Check Qxxx.x German' | French: 'S3 250 Row 26 Failed To Advance.. Check Qxxx.x French'
  251 = 'S3 251 Row 26 Failed To Return.. Check Qxxx.x Default' | German: 'S3 251 Row 26 Failed To Return.. Check Qxxx.x German' | French: 'S3 251 Row 26 Failed To Return.. Check Qxxx.x French'
  252 = 'S3 252 Row 26 Lost Advance Position... Check Ixxx.x Default' | German: 'S3 252 Row 26 Lost Advance Position... Check Ixxx.x German' | French: 'S3 252 Row 26 Lost Advance Position... Check Ixxx.x French'
  253 = 'S3 253 Row 26 Lost Return Position... Check Ixxx.x Default' | German: 'S3 253 Row 26 Lost Return Position... Check Ixxx.x German' | French: 'S3 253 Row 26 Lost Return Position... Check Ixxx.x French'
  254 = 'S3 254 Row 26 Switch Fault... Check Ixxx.x / Ixxx.x Default' | German: 'S3 254 Row 26 Switch Fault... Check Ixxx.x / Ixxx.x German' | French: 'S3 254 Row 26 Switch Fault... Check Ixxx.x / Ixxx.x French'
  255 = 'S3 255 Row 26 Spare Message Default' | German: 'S3 255 Row 26 Spare Message German' | French: 'S3 255 Row 26 Spare Message French'
  256 = 'S3 256 Row 26 Spare Message Default' | German: 'S3 256 Row 26 Spare Message German' | French: 'S3 256 Row 26 Spare Message French'
  257 = 'S3 257 Row 26 Spare Message Default' | German: 'S3 257 Row 26 Spare Message German' | French: 'S3 257 Row 26 Spare Message French'
  258 = 'S3 258 Row 26 Spare Message Default' | German: 'S3 258 Row 26 Spare Message German' | French: 'S3 258 Row 26 Spare Message French'
  259 = 'S3 259 Row 26 Spare Message Default' | German: 'S3 259 Row 26 Spare Message German' | French: 'S3 259 Row 26 Spare Message French'
  260 = 'S3 260 Row 27 Failed To Advance.. Check Qxxx.x Default' | German: 'S3 260 Row 27 Failed To Advance.. Check Qxxx.x German' | French: 'S3 260 Row 27 Failed To Advance.. Check Qxxx.x French'
  261 = 'S3 261 Row 27 Failed To Return.. Check Qxxx.x Default' | German: 'S3 261 Row 27 Failed To Return.. Check Qxxx.x German' | French: 'S3 261 Row 27 Failed To Return.. Check Qxxx.x French'
  262 = 'S3 262 Row 27 Lost Advance Position... Check Ixxx.x Default' | German: 'S3 262 Row 27 Lost Advance Position... Check Ixxx.x German' | French: 'S3 262 Row 27 Lost Advance Position... Check Ixxx.x French'
  263 = 'S3 263 Row 27 Lost Return Position... Check Ixxx.x Default' | German: 'S3 263 Row 27 Lost Return Position... Check Ixxx.x German' | French: 'S3 263 Row 27 Lost Return Position... Check Ixxx.x French'
  264 = 'S3 264 Row 27 Switch Fault... Check Ixxx.x / Ixxx.x Default' | German: 'S3 264 Row 27 Switch Fault... Check Ixxx.x / Ixxx.x German' | French: 'S3 264 Row 27 Switch Fault... Check Ixxx.x / Ixxx.x French'
  265 = 'S3 265 Row 27 Spare Message Default' | German: 'S3 265 Row 27 Spare Message German' | French: 'S3 265 Row 27 Spare Message French'
  266 = 'S3 266 Row 27 Spare Message Default' | German: 'S3 266 Row 27 Spare Message German' | French: 'S3 266 Row 27 Spare Message French'
  267 = 'S3 267 Row 27 Spare Message Default' | German: 'S3 267 Row 27 Spare Message German' | French: 'S3 267 Row 27 Spare Message French'
  268 = 'S3 268 Row 27 Spare Message Default' | German: 'S3 268 Row 27 Spare Message German' | French: 'S3 268 Row 27 Spare Message French'
  269 = 'S3 269 Row 27 Spare Message Default' | German: 'S3 269 Row 27 Spare Message German' | French: 'S3 269 Row 27 Spare Message French'
  270 = 'S3 270 Row 28 Failed To Advance.. Check Qxxx.x Default' | German: 'S3 270 Row 28 Failed To Advance.. Check Qxxx.x German' | French: 'S3 270 Row 28 Failed To Advance.. Check Qxxx.x French'
  271 = 'S3 271 Row 28 Failed To Return.. Check Qxxx.x Default' | German: 'S3 271 Row 28 Failed To Return.. Check Qxxx.x German' | French: 'S3 271 Row 28 Failed To Return.. Check Qxxx.x French'
  272 = 'S3 272 Row 28 Lost Advance Position... Check Ixxx.x Default' | German: 'S3 272 Row 28 Lost Advance Position... Check Ixxx.x German' | French: 'S3 272 Row 28 Lost Advance Position... Check Ixxx.x French'
  273 = 'S3 273 Row 28 Lost Return Position... Check Ixxx.x Default' | German: 'S3 273 Row 28 Lost Return Position... Check Ixxx.x German' | French: 'S3 273 Row 28 Lost Return Position... Check Ixxx.x French'
  274 = 'S3 274 Row 28 Switch Fault... Check Ixxx.x / Ixxx.x Default' | German: 'S3 274 Row 28 Switch Fault... Check Ixxx.x / Ixxx.x German' | French: 'S3 274 Row 28 Switch Fault... Check Ixxx.x / Ixxx.x French'
  275 = 'S3 275 Row 28 Spare Message Default' | German: 'S3 275 Row 28 Spare Message German' | French: 'S3 275 Row 28 Spare Message French'
  276 = 'S3 276 Row 28 Spare Message Default' | German: 'S3 276 Row 28 Spare Message German' | French: 'S3 276 Row 28 Spare Message French'
  277 = 'S3 277 Row 28 Spare Message Default' | German: 'S3 277 Row 28 Spare Message German' | French: 'S3 277 Row 28 Spare Message French'
  278 = 'S3 278 Row 28 Spare Message Default' | German: 'S3 278 Row 28 Spare Message German' | French: 'S3 278 Row 28 Spare Message French'
  279 = 'S3 279 Row 28 Spare Message Default' | German: 'S3 279 Row 28 Spare Message German' | French: 'S3 279 Row 28 Spare Message French'
  280 = 'S3 280 Row 29 Failed To Advance.. Check Qxxx.x Default' | German: 'S3 280 Row 29 Failed To Advance.. Check Qxxx.x German' | French: 'S3 280 Row 29 Failed To Advance.. Check Qxxx.x French'
  281 = 'S3 281 Row 29 Failed To Return.. Check Qxxx.x Default' | German: 'S3 281 Row 29 Failed To Return.. Check Qxxx.x German' | French: 'S3 281 Row 29 Failed To Return.. Check Qxxx.x French'
  282 = 'S3 282 Row 29 Lost Advance Position... Check Ixxx.x Default' | German: 'S3 282 Row 29 Lost Advance Position... Check Ixxx.x German' | French: 'S3 282 Row 29 Lost Advance Position... Check Ixxx.x French'
  283 = 'S3 283 Row 29 Lost Return Position... Check Ixxx.x Default' | German: 'S3 283 Row 29 Lost Return Position... Check Ixxx.x German' | French: 'S3 283 Row 29 Lost Return Position... Check Ixxx.x French'
  284 = 'S3 284 Row 29 Switch Fault... Check Ixxx.x / Ixxx.x Default' | German: 'S3 284 Row 29 Switch Fault... Check Ixxx.x / Ixxx.x German' | French: 'S3 284 Row 29 Switch Fault... Check Ixxx.x / Ixxx.x French'
  285 = 'S3 285 Row 29 Spare Message Default' | German: 'S3 285 Row 29 Spare Message German' | French: 'S3 285 Row 29 Spare Message French'
  286 = 'S3 286 Row 29 Spare Message Default' | German: 'S3 286 Row 29 Spare Message German' | French: 'S3 286 Row 29 Spare Message French'
  287 = 'S3 287 Row 29 Spare Message Default' | German: 'S3 287 Row 29 Spare Message German' | French: 'S3 287 Row 29 Spare Message French'
  288 = 'S3 288 Row 29 Spare Message Default' | German: 'S3 288 Row 29 Spare Message German' | French: 'S3 288 Row 29 Spare Message French'
  289 = 'S3 289 Row 29 Spare Message Default' | German: 'S3 289 Row 29 Spare Message German' | French: 'S3 289 Row 29 Spare Message French'
  290 = 'S3 290 Row 30 Failed To Advance.. Check Qxxx.x Default' | German: 'S3 290 Row 30 Failed To Advance.. Check Qxxx.x German' | French: 'S3 290 Row 30 Failed To Advance.. Check Qxxx.x French'
  291 = 'S3 291 Row 30 Failed To Return.. Check Qxxx.x Default' | German: 'S3 291 Row 30 Failed To Return.. Check Qxxx.x German' | French: 'S3 291 Row 30 Failed To Return.. Check Qxxx.x French'
  292 = 'S3 292 Row 30 Lost Advance Position... Check Ixxx.x Default' | German: 'S3 292 Row 30 Lost Advance Position... Check Ixxx.x German' | French: 'S3 292 Row 30 Lost Advance Position... Check Ixxx.x French'
  293 = 'S3 293 Row 30 Lost Return Position... Check Ixxx.x Default' | German: 'S3 293 Row 30 Lost Return Position... Check Ixxx.x German' | French: 'S3 293 Row 30 Lost Return Position... Check Ixxx.x French'
  294 = 'S3 294 Row 30 Switch Fault... Check Ixxx.x / Ixxx.x Default' | German: 'S3 294 Row 30 Switch Fault... Check Ixxx.x / Ixxx.x German' | French: 'S3 294 Row 30 Switch Fault... Check Ixxx.x / Ixxx.x French'
  295 = 'S3 295 Row 30 Spare Message Default' | German: 'S3 295 Row 30 Spare Message German' | French: 'S3 295 Row 30 Spare Message French'
  296 = 'S3 296 Row 30 Spare Message Default' | German: 'S3 296 Row 30 Spare Message German' | French: 'S3 296 Row 30 Spare Message French'
  297 = 'S3 297 Row 30 Spare Message Default' | German: 'S3 297 Row 30 Spare Message German' | French: 'S3 297 Row 30 Spare Message French'
  298 = 'S3 298 Row 30 Spare Message Default' | German: 'S3 298 Row 30 Spare Message German' | French: 'S3 298 Row 30 Spare Message French'
  299 = 'S3 299 Row 30 Spare Message Default' | German: 'S3 299 Row 30 Spare Message German' | French: 'S3 299 Row 30 Spare Message French'
  300 = 'S3 300 Row 31 Failed To Advance.. Check Qxxx.x Default' | German: 'S3 300 Row 31 Failed To Advance.. Check Qxxx.x German' | French: 'S3 300 Row 31 Failed To Advance.. Check Qxxx.x French'
  301 = 'S3 301 Row 31 Failed To Return.. Check Qxxx.x Default' | German: 'S3 301 Row 31 Failed To Return.. Check Qxxx.x German' | French: 'S3 301 Row 31 Failed To Return.. Check Qxxx.x French'
  302 = 'S3 302 Row 31 Lost Advance Position... Check Ixxx.x Default' | German: 'S3 302 Row 31 Lost Advance Position... Check Ixxx.x German' | French: 'S3 302 Row 31 Lost Advance Position... Check Ixxx.x French'
  303 = 'S3 303 Row 31 Lost Return Position... Check Ixxx.x Default' | German: 'S3 303 Row 31 Lost Return Position... Check Ixxx.x German' | French: 'S3 303 Row 31 Lost Return Position... Check Ixxx.x French'
  304 = 'S3 304 Row 31 Switch Fault... Check Ixxx.x / Ixxx.x Default' | German: 'S3 304 Row 31 Switch Fault... Check Ixxx.x / Ixxx.x German' | French: 'S3 304 Row 31 Switch Fault... Check Ixxx.x / Ixxx.x French'
  305 = 'S3 305 Row 31 Spare Message Default' | German: 'S3 305 Row 31 Spare Message German' | French: 'S3 305 Row 31 Spare Message French'
  306 = 'S3 306 Row 31 Spare Message Default' | German: 'S3 306 Row 31 Spare Message German' | French: 'S3 306 Row 31 Spare Message French'
  307 = 'S3 307 Row 31 Spare Message Default' | German: 'S3 307 Row 31 Spare Message German' | French: 'S3 307 Row 31 Spare Message French'
  308 = 'S3 308 Row 31 Spare Message Default' | German: 'S3 308 Row 31 Spare Message German' | French: 'S3 308 Row 31 Spare Message French'
  309 = 'S3 309 Row 31 Spare Message Default' | German: 'S3 309 Row 31 Spare Message German' | French: 'S3 309 Row 31 Spare Message French'
  310 = 'S3 310 Row 32 Failed To Advance.. Check Qxxx.x Default' | German: 'S3 310 Row 32 Failed To Advance.. Check Qxxx.x German' | French: 'S3 310 Row 32 Failed To Advance.. Check Qxxx.x French'
  311 = 'S3 311 Row 32 Failed To Return.. Check Qxxx.x Default' | German: 'S3 311 Row 32 Failed To Return.. Check Qxxx.x German' | French: 'S3 311 Row 32 Failed To Return.. Check Qxxx.x French'
  312 = 'S3 312 Row 32 Lost Advance Position... Check Ixxx.x Default' | German: 'S3 312 Row 32 Lost Advance Position... Check Ixxx.x German' | French: 'S3 312 Row 32 Lost Advance Position... Check Ixxx.x French'
  313 = 'S3 313 Row 32 Lost Return Position... Check Ixxx.x Default' | German: 'S3 313 Row 32 Lost Return Position... Check Ixxx.x German' | French: 'S3 313 Row 32 Lost Return Position... Check Ixxx.x French'
  314 = 'S3 314 Row 32 Switch Fault... Check Ixxx.x / Ixxx.x Default' | German: 'S3 314 Row 32 Switch Fault... Check Ixxx.x / Ixxx.x German' | French: 'S3 314 Row 32 Switch Fault... Check Ixxx.x / Ixxx.x French'
  315 = 'S3 315 Row 32 Spare Message Default' | German: 'S3 315 Row 32 Spare Message German' | French: 'S3 315 Row 32 Spare Message French'
  316 = 'S3 316 Row 32 Spare Message Default' | German: 'S3 316 Row 32 Spare Message German' | French: 'S3 316 Row 32 Spare Message French'
  317 = 'S3 317 Row 32 Spare Message Default' | German: 'S3 317 Row 32 Spare Message German' | French: 'S3 317 Row 32 Spare Message French'
  318 = 'S3 318 Row 32 Spare Message Default' | German: 'S3 318 Row 32 Spare Message German' | French: 'S3 318 Row 32 Spare Message French'
  319 = 'S3 319 Row 32 Spare Message Default' | German: 'S3 319 Row 32 Spare Message German' | French: 'S3 319 Row 32 Spare Message French'
  320 = 'S3 320 Row 33 Failed To Advance.. Check Qxxx.x Default' | German: 'S3 320 Row 33 Failed To Advance.. Check Qxxx.x German' | French: 'S3 320 Row 33 Failed To Advance.. Check Qxxx.x French'
  321 = 'S3 321 Row 33 Failed To Return.. Check Qxxx.x Default' | German: 'S3 321 Row 33 Failed To Return.. Check Qxxx.x German' | French: 'S3 321 Row 33 Failed To Return.. Check Qxxx.x French'
  322 = 'S3 322 Row 33 Lost Advance Position... Check Ixxx.x Default' | German: 'S3 322 Row 33 Lost Advance Position... Check Ixxx.x German' | French: 'S3 322 Row 33 Lost Advance Position... Check Ixxx.x French'
  323 = 'S3 323 Row 33 Lost Return Position... Check Ixxx.x Default' | German: 'S3 323 Row 33 Lost Return Position... Check Ixxx.x German' | French: 'S3 323 Row 33 Lost Return Position... Check Ixxx.x French'
  324 = 'S3 324 Row 33 Switch Fault... Check Ixxx.x / Ixxx.x Default' | German: 'S3 324 Row 33 Switch Fault... Check Ixxx.x / Ixxx.x German' | French: 'S3 324 Row 33 Switch Fault... Check Ixxx.x / Ixxx.x French'
  325 = 'S3 325 Row 33 Spare Message Default' | German: 'S3 325 Row 33 Spare Message German' | French: 'S3 325 Row 33 Spare Message French'
  326 = 'S3 326 Row 33 Spare Message Default' | German: 'S3 326 Row 33 Spare Message German' | French: 'S3 326 Row 33 Spare Message French'
  327 = 'S3 327 Row 33 Spare Message Default' | German: 'S3 327 Row 33 Spare Message German' | French: 'S3 327 Row 33 Spare Message French'
  328 = 'S3 328 Row 33 Spare Message Default' | German: 'S3 328 Row 33 Spare Message German' | French: 'S3 328 Row 33 Spare Message French'
  329 = 'S3 329 Row 33 Spare Message Default' | German: 'S3 329 Row 33 Spare Message German' | French: 'S3 329 Row 33 Spare Message French'
  330 = 'S3 330 Row 34 Failed To Advance.. Check Qxxx.x Default' | German: 'S3 330 Row 34 Failed To Advance.. Check Qxxx.x German' | French: 'S3 330 Row 34 Failed To Advance.. Check Qxxx.x French'
  331 = 'S3 331 Row 34 Failed To Return.. Check Qxxx.x Default' | German: 'S3 331 Row 34 Failed To Return.. Check Qxxx.x German' | French: 'S3 331 Row 34 Failed To Return.. Check Qxxx.x French'
  332 = 'S3 332 Row 34 Lost Advance Position... Check Ixxx.x Default' | German: 'S3 332 Row 34 Lost Advance Position... Check Ixxx.x German' | French: 'S3 332 Row 34 Lost Advance Position... Check Ixxx.x French'
  333 = 'S3 333 Row 34 Lost Return Position... Check Ixxx.x Default' | German: 'S3 333 Row 34 Lost Return Position... Check Ixxx.x German' | French: 'S3 333 Row 34 Lost Return Position... Check Ixxx.x French'
  334 = 'S3 334 Row 34 Switch Fault... Check Ixxx.x / Ixxx.x Default' | German: 'S3 334 Row 34 Switch Fault... Check Ixxx.x / Ixxx.x German' | French: 'S3 334 Row 34 Switch Fault... Check Ixxx.x / Ixxx.x French'
  335 = 'S3 335 Row 34 Spare Message Default' | German: 'S3 335 Row 34 Spare Message German' | French: 'S3 335 Row 34 Spare Message French'
  336 = 'S3 336 Row 34 Spare Message Default' | German: 'S3 336 Row 34 Spare Message German' | French: 'S3 336 Row 34 Spare Message French'
  337 = 'S3 337 Row 34 Spare Message Default' | German: 'S3 337 Row 34 Spare Message German' | French: 'S3 337 Row 34 Spare Message French'
  338 = 'S3 338 Row 34 Spare Message Default' | German: 'S3 338 Row 34 Spare Message German' | French: 'S3 338 Row 34 Spare Message French'
  339 = 'S3 339 Row 34 Spare Message Default' | German: 'S3 339 Row 34 Spare Message German' | French: 'S3 339 Row 34 Spare Message French'
  340 = 'S3 340 Row 35 Failed To Advance.. Check Qxxx.x Default' | German: 'S3 340 Row 35 Failed To Advance.. Check Qxxx.x German' | French: 'S3 340 Row 35 Failed To Advance.. Check Qxxx.x French'
  341 = 'S3 341 Row 35 Failed To Return.. Check Qxxx.x Default' | German: 'S3 341 Row 35 Failed To Return.. Check Qxxx.x German' | French: 'S3 341 Row 35 Failed To Return.. Check Qxxx.x French'
  342 = 'S3 342 Row 35 Lost Advance Position... Check Ixxx.x Default' | German: 'S3 342 Row 35 Lost Advance Position... Check Ixxx.x German' | French: 'S3 342 Row 35 Lost Advance Position... Check Ixxx.x French'
  343 = 'S3 343 Row 35 Lost Return Position... Check Ixxx.x Default' | German: 'S3 343 Row 35 Lost Return Position... Check Ixxx.x German' | French: 'S3 343 Row 35 Lost Return Position... Check Ixxx.x French'
  344 = 'S3 344 Row 35 Switch Fault... Check Ixxx.x / Ixxx.x Default' | German: 'S3 344 Row 35 Switch Fault... Check Ixxx.x / Ixxx.x German' | French: 'S3 344 Row 35 Switch Fault... Check Ixxx.x / Ixxx.x French'
  345 = 'S3 345 Row 35 Spare Message Default' | German: 'S3 345 Row 35 Spare Message German' | French: 'S3 345 Row 35 Spare Message French'
  346 = 'S3 346 Row 35 Spare Message Default' | German: 'S3 346 Row 35 Spare Message German' | French: 'S3 346 Row 35 Spare Message French'
  347 = 'S3 347 Row 35 Spare Message Default' | German: 'S3 347 Row 35 Spare Message German' | French: 'S3 347 Row 35 Spare Message French'
  348 = 'S3 348 Row 35 Spare Message Default' | German: 'S3 348 Row 35 Spare Message German' | French: 'S3 348 Row 35 Spare Message French'
  349 = 'S3 349 Row 35 Spare Message Default' | German: 'S3 349 Row 35 Spare Message German' | French: 'S3 349 Row 35 Spare Message French'
  350 = 'S3 350 Row 36 Failed To Advance.. Check Qxxx.x Default' | German: 'S3 350 Row 36 Failed To Advance.. Check Qxxx.x German' | French: 'S3 350 Row 36 Failed To Advance.. Check Qxxx.x French'
  351 = 'S3 351 Row 36 Failed To Return.. Check Qxxx.x Default' | German: 'S3 351 Row 36 Failed To Return.. Check Qxxx.x German' | French: 'S3 351 Row 36 Failed To Return.. Check Qxxx.x French'
  352 = 'S3 352 Row 36 Lost Advance Position... Check Ixxx.x Default' | German: 'S3 352 Row 36 Lost Advance Position... Check Ixxx.x German' | French: 'S3 352 Row 36 Lost Advance Position... Check Ixxx.x French'
  353 = 'S3 353 Row 36 Lost Return Position... Check Ixxx.x Default' | German: 'S3 353 Row 36 Lost Return Position... Check Ixxx.x German' | French: 'S3 353 Row 36 Lost Return Position... Check Ixxx.x French'
  354 = 'S3 354 Row 36 Switch Fault... Check Ixxx.x / Ixxx.x Default' | German: 'S3 354 Row 36 Switch Fault... Check Ixxx.x / Ixxx.x German' | French: 'S3 354 Row 36 Switch Fault... Check Ixxx.x / Ixxx.x French'
  355 = 'S3 355 Row 36 Spare Message Default' | German: 'S3 355 Row 36 Spare Message German' | French: 'S3 355 Row 36 Spare Message French'
  356 = 'S3 356 Row 36 Spare Message Default' | German: 'S3 356 Row 36 Spare Message German' | French: 'S3 356 Row 36 Spare Message French'
  357 = 'S3 357 Row 36 Spare Message Default' | German: 'S3 357 Row 36 Spare Message German' | French: 'S3 357 Row 36 Spare Message French'
  358 = 'S3 358 Row 36 Spare Message Default' | German: 'S3 358 Row 36 Spare Message German' | French: 'S3 358 Row 36 Spare Message French'
  359 = 'S3 359 Row 36 Spare Message Default' | German: 'S3 359 Row 36 Spare Message German' | French: 'S3 359 Row 36 Spare Message French'
  360 = 'S3 360 Row 37 Failed To Advance.. Check Qxxx.x Default' | German: 'S3 360 Row 37 Failed To Advance.. Check Qxxx.x German' | French: 'S3 360 Row 37 Failed To Advance.. Check Qxxx.x French'
  361 = 'S3 361 Row 37 Failed To Return.. Check Qxxx.x Default' | German: 'S3 361 Row 37 Failed To Return.. Check Qxxx.x German' | French: 'S3 361 Row 37 Failed To Return.. Check Qxxx.x French'
  362 = 'S3 362 Row 37 Lost Advance Position... Check Ixxx.x Default' | German: 'S3 362 Row 37 Lost Advance Position... Check Ixxx.x German' | French: 'S3 362 Row 37 Lost Advance Position... Check Ixxx.x French'
  363 = 'S3 363 Row 37 Lost Return Position... Check Ixxx.x Default' | German: 'S3 363 Row 37 Lost Return Position... Check Ixxx.x German' | French: 'S3 363 Row 37 Lost Return Position... Check Ixxx.x French'
  364 = 'S3 364 Row 37 Switch Fault... Check Ixxx.x / Ixxx.x Default' | German: 'S3 364 Row 37 Switch Fault... Check Ixxx.x / Ixxx.x German' | French: 'S3 364 Row 37 Switch Fault... Check Ixxx.x / Ixxx.x French'
  365 = 'S3 365 Row 37 Spare Message Default' | German: 'S3 365 Row 37 Spare Message German' | French: 'S3 365 Row 37 Spare Message French'
  366 = 'S3 366 Row 37 Spare Message Default' | German: 'S3 366 Row 37 Spare Message German' | French: 'S3 366 Row 37 Spare Message French'
  367 = 'S3 367 Row 37 Spare Message Default' | German: 'S3 367 Row 37 Spare Message German' | French: 'S3 367 Row 37 Spare Message French'
  368 = 'S3 368 Row 37 Spare Message Default' | German: 'S3 368 Row 37 Spare Message German' | French: 'S3 368 Row 37 Spare Message French'
  369 = 'S3 369 Row 37 Spare Message Default' | German: 'S3 369 Row 37 Spare Message German' | French: 'S3 369 Row 37 Spare Message French'
  370 = 'S3 370 Row 38 Failed To Advance.. Check Qxxx.x Default' | German: 'S3 370 Row 38 Failed To Advance.. Check Qxxx.x German' | French: 'S3 370 Row 38 Failed To Advance.. Check Qxxx.x French'
  371 = 'S3 371 Row 38 Failed To Return.. Check Qxxx.x Default' | German: 'S3 371 Row 38 Failed To Return.. Check Qxxx.x German' | French: 'S3 371 Row 38 Failed To Return.. Check Qxxx.x French'
  372 = 'S3 372 Row 38 Lost Advance Position... Check Ixxx.x Default' | German: 'S3 372 Row 38 Lost Advance Position... Check Ixxx.x German' | French: 'S3 372 Row 38 Lost Advance Position... Check Ixxx.x French'
  373 = 'S3 373 Row 38 Lost Return Position... Check Ixxx.x Default' | German: 'S3 373 Row 38 Lost Return Position... Check Ixxx.x German' | French: 'S3 373 Row 38 Lost Return Position... Check Ixxx.x French'
  374 = 'S3 374 Row 38 Switch Fault... Check Ixxx.x / Ixxx.x Default' | German: 'S3 374 Row 38 Switch Fault... Check Ixxx.x / Ixxx.x German' | French: 'S3 374 Row 38 Switch Fault... Check Ixxx.x / Ixxx.x French'
  375 = 'S3 375 Row 38 Spare Message Default' | German: 'S3 375 Row 38 Spare Message German' | French: 'S3 375 Row 38 Spare Message French'
  376 = 'S3 376 Row 38 Spare Message Default' | German: 'S3 376 Row 38 Spare Message German' | French: 'S3 376 Row 38 Spare Message French'
  377 = 'S3 377 Row 38 Spare Message Default' | German: 'S3 377 Row 38 Spare Message German' | French: 'S3 377 Row 38 Spare Message French'
  378 = 'S3 378 Row 38 Spare Message Default' | German: 'S3 378 Row 38 Spare Message German' | French: 'S3 378 Row 38 Spare Message French'
  379 = 'S3 379 Row 38 Spare Message Default' | German: 'S3 379 Row 38 Spare Message German' | French: 'S3 379 Row 38 Spare Message French'
  380 = 'S3 380 Row 39 Failed To Advance.. Check Qxxx.x Default' | German: 'S3 380 Row 39 Failed To Advance.. Check Qxxx.x German' | French: 'S3 380 Row 39 Failed To Advance.. Check Qxxx.x French'
  381 = 'S3 381 Row 39 Failed To Return.. Check Qxxx.x Default' | German: 'S3 381 Row 39 Failed To Return.. Check Qxxx.x German' | French: 'S3 381 Row 39 Failed To Return.. Check Qxxx.x French'
  382 = 'S3 382 Row 39 Lost Advance Position... Check Ixxx.x Default' | German: 'S3 382 Row 39 Lost Advance Position... Check Ixxx.x German' | French: 'S3 382 Row 39 Lost Advance Position... Check Ixxx.x French'
  383 = 'S3 383 Row 39 Lost Return Position... Check Ixxx.x Default' | German: 'S3 383 Row 39 Lost Return Position... Check Ixxx.x German' | French: 'S3 383 Row 39 Lost Return Position... Check Ixxx.x French'
  384 = 'S3 384 Row 39 Switch Fault... Check Ixxx.x / Ixxx.x Default' | German: 'S3 384 Row 39 Switch Fault... Check Ixxx.x / Ixxx.x German' | French: 'S3 384 Row 39 Switch Fault... Check Ixxx.x / Ixxx.x French'
  385 = 'S3 385 Row 39 Spare Message Default' | German: 'S3 385 Row 39 Spare Message German' | French: 'S3 385 Row 39 Spare Message French'
  386 = 'S3 386 Row 39 Spare Message Default' | German: 'S3 386 Row 39 Spare Message German' | French: 'S3 386 Row 39 Spare Message French'
  387 = 'S3 387 Row 39 Spare Message Default' | German: 'S3 387 Row 39 Spare Message German' | French: 'S3 387 Row 39 Spare Message French'
  388 = 'S3 388 Row 39 Spare Message Default' | German: 'S3 388 Row 39 Spare Message German' | French: 'S3 388 Row 39 Spare Message French'
  389 = 'S3 389 Row 39 Spare Message Default' | German: 'S3 389 Row 39 Spare Message German' | French: 'S3 389 Row 39 Spare Message French'
  390 = 'S3 390 Row 40 Failed To Advance.. Check Qxxx.x Default' | German: 'S3 390 Row 40 Failed To Advance.. Check Qxxx.x German' | French: 'S3 390 Row 40 Failed To Advance.. Check Qxxx.x French'
  391 = 'S3 391 Row 40 Failed To Return.. Check Qxxx.x Default' | German: 'S3 391 Row 40 Failed To Return.. Check Qxxx.x German' | French: 'S3 391 Row 40 Failed To Return.. Check Qxxx.x French'
  392 = 'S3 392 Row 40 Lost Advance Position... Check Ixxx.x Default' | German: 'S3 392 Row 40 Lost Advance Position... Check Ixxx.x German' | French: 'S3 392 Row 40 Lost Advance Position... Check Ixxx.x French'
  393 = 'S3 393 Row 40 Lost Return Position... Check Ixxx.x Default' | German: 'S3 393 Row 40 Lost Return Position... Check Ixxx.x German' | French: 'S3 393 Row 40 Lost Return Position... Check Ixxx.x French'
  394 = 'S3 394 Row 40 Switch Fault... Check Ixxx.x / Ixxx.x Default' | German: 'S3 394 Row 40 Switch Fault... Check Ixxx.x / Ixxx.x German' | French: 'S3 394 Row 40 Switch Fault... Check Ixxx.x / Ixxx.x French'
  395 = 'S3 395 Row 40 Spare Message Default' | German: 'S3 395 Row 40 Spare Message German' | French: 'S3 395 Row 40 Spare Message French'
  396 = 'S3 396 Row 40 Spare Message Default' | German: 'S3 396 Row 40 Spare Message German' | French: 'S3 396 Row 40 Spare Message French'
  397 = 'S3 397 Row 40 Spare Message Default' | German: 'S3 397 Row 40 Spare Message German' | French: 'S3 397 Row 40 Spare Message French'
  398 = 'S3 398 Row 40 Spare Message Default' | German: 'S3 398 Row 40 Spare Message German' | French: 'S3 398 Row 40 Spare Message French'
  399 = 'S3 399 Row 40 Spare Message Default' | German: 'S3 399 Row 40 Spare Message German' | French: 'S3 399 Row 40 Spare Message French'
  400 = 'S3 400 Row 41 Failed To Advance.. Check Qxxx.x Default' | German: 'S3 400 Row 41 Failed To Advance.. Check Qxxx.x German' | French: 'S3 400 Row 41 Failed To Advance.. Check Qxxx.x French'
  401 = 'S3 401 Row 41 Failed To Return.. Check Qxxx.x Default' | German: 'S3 401 Row 41 Failed To Return.. Check Qxxx.x German' | French: 'S3 401 Row 41 Failed To Return.. Check Qxxx.x French'
  402 = 'S3 402 Row 41 Lost Advance Position... Check Ixxx.x Default' | German: 'S3 402 Row 41 Lost Advance Position... Check Ixxx.x German' | French: 'S3 402 Row 41 Lost Advance Position... Check Ixxx.x French'
  403 = 'S3 403 Row 41 Lost Return Position... Check Ixxx.x Default' | German: 'S3 403 Row 41 Lost Return Position... Check Ixxx.x German' | French: 'S3 403 Row 41 Lost Return Position... Check Ixxx.x French'
  404 = 'S3 404 Row 41 Switch Fault... Check Ixxx.x / Ixxx.x Default' | German: 'S3 404 Row 41 Switch Fault... Check Ixxx.x / Ixxx.x German' | French: 'S3 404 Row 41 Switch Fault... Check Ixxx.x / Ixxx.x French'
  405 = 'S3 405 Row 41 Spare Message Default' | German: 'S3 405 Row 41 Spare Message German' | French: 'S3 405 Row 41 Spare Message French'
  406 = 'S3 406 Row 41 Spare Message Default' | German: 'S3 406 Row 41 Spare Message German' | French: 'S3 406 Row 41 Spare Message French'
  407 = 'S3 407 Row 41 Spare Message Default' | German: 'S3 407 Row 41 Spare Message German' | French: 'S3 407 Row 41 Spare Message French'
  408 = 'S3 408 Row 41 Spare Message Default' | German: 'S3 408 Row 41 Spare Message German' | French: 'S3 408 Row 41 Spare Message French'
  409 = 'S3 409 Row 41 Spare Message Default' | German: 'S3 409 Row 41 Spare Message German' | French: 'S3 409 Row 41 Spare Message French'
  410 = 'S3 410 Row 42 Failed To Advance.. Check Qxxx.x Default' | German: 'S3 410 Row 42 Failed To Advance.. Check Qxxx.x German' | French: 'S3 410 Row 42 Failed To Advance.. Check Qxxx.x French'
  411 = 'S3 411 Row 42 Failed To Return.. Check Qxxx.x Default' | German: 'S3 411 Row 42 Failed To Return.. Check Qxxx.x German' | French: 'S3 411 Row 42 Failed To Return.. Check Qxxx.x French'
  412 = 'S3 412 Row 42 Lost Advance Position... Check Ixxx.x Default' | German: 'S3 412 Row 42 Lost Advance Position... Check Ixxx.x German' | French: 'S3 412 Row 42 Lost Advance Position... Check Ixxx.x French'
  413 = 'S3 413 Row 42 Lost Return Position... Check Ixxx.x Default' | German: 'S3 413 Row 42 Lost Return Position... Check Ixxx.x German' | French: 'S3 413 Row 42 Lost Return Position... Check Ixxx.x French'
  414 = 'S3 414 Row 42 Switch Fault... Check Ixxx.x / Ixxx.x Default' | German: 'S3 414 Row 42 Switch Fault... Check Ixxx.x / Ixxx.x German' | French: 'S3 414 Row 42 Switch Fault... Check Ixxx.x / Ixxx.x French'
  415 = 'S3 415 Row 42 Spare Message Default' | German: 'S3 415 Row 42 Spare Message German' | French: 'S3 415 Row 42 Spare Message French'
  416 = 'S3 416 Row 42 Spare Message Default' | German: 'S3 416 Row 42 Spare Message German' | French: 'S3 416 Row 42 Spare Message French'
  417 = 'S3 417 Row 42 Spare Message Default' | German: 'S3 417 Row 42 Spare Message German' | French: 'S3 417 Row 42 Spare Message French'
  418 = 'S3 418 Row 42 Spare Message Default' | German: 'S3 418 Row 42 Spare Message German' | French: 'S3 418 Row 42 Spare Message French'
  419 = 'S3 419 Row 42 Spare Message Default' | German: 'S3 419 Row 42 Spare Message German' | French: 'S3 419 Row 42 Spare Message French'
  420 = 'S3 420 Row 43 Failed To Advance.. Check Qxxx.x Default' | German: 'S3 420 Row 43 Failed To Advance.. Check Qxxx.x German' | French: 'S3 420 Row 43 Failed To Advance.. Check Qxxx.x French'
  421 = 'S3 421 Row 43 Failed To Return.. Check Qxxx.x Default' | German: 'S3 421 Row 43 Failed To Return.. Check Qxxx.x German' | French: 'S3 421 Row 43 Failed To Return.. Check Qxxx.x French'
  422 = 'S3 422 Row 43 Lost Advance Position... Check Ixxx.x Default' | German: 'S3 422 Row 43 Lost Advance Position... Check Ixxx.x German' | French: 'S3 422 Row 43 Lost Advance Position... Check Ixxx.x French'
  423 = 'S3 423 Row 43 Lost Return Position... Check Ixxx.x Default' | German: 'S3 423 Row 43 Lost Return Position... Check Ixxx.x German' | French: 'S3 423 Row 43 Lost Return Position... Check Ixxx.x French'
  424 = 'S3 424 Row 43 Switch Fault... Check Ixxx.x / Ixxx.x Default' | German: 'S3 424 Row 43 Switch Fault... Check Ixxx.x / Ixxx.x German' | French: 'S3 424 Row 43 Switch Fault... Check Ixxx.x / Ixxx.x French'
  425 = 'S3 425 Row 43 Spare Message Default' | German: 'S3 425 Row 43 Spare Message German' | French: 'S3 425 Row 43 Spare Message French'
  426 = 'S3 426 Row 43 Spare Message Default' | German: 'S3 426 Row 43 Spare Message German' | French: 'S3 426 Row 43 Spare Message French'
  427 = 'S3 427 Row 43 Spare Message Default' | German: 'S3 427 Row 43 Spare Message German' | French: 'S3 427 Row 43 Spare Message French'
  428 = 'S3 428 Row 43 Spare Message Default' | German: 'S3 428 Row 43 Spare Message German' | French: 'S3 428 Row 43 Spare Message French'
  429 = 'S3 429 Row 43 Spare Message Default' | German: 'S3 429 Row 43 Spare Message German' | French: 'S3 429 Row 43 Spare Message French'
  430 = 'S3 430 Row 44 Failed To Advance.. Check Qxxx.x Default' | German: 'S3 430 Row 44 Failed To Advance.. Check Qxxx.x German' | French: 'S3 430 Row 44 Failed To Advance.. Check Qxxx.x French'
  431 = 'S3 431 Row 44 Failed To Return.. Check Qxxx.x Default' | German: 'S3 431 Row 44 Failed To Return.. Check Qxxx.x German' | French: 'S3 431 Row 44 Failed To Return.. Check Qxxx.x French'
  432 = 'S3 432 Row 44 Lost Advance Position... Check Ixxx.x Default' | German: 'S3 432 Row 44 Lost Advance Position... Check Ixxx.x German' | French: 'S3 432 Row 44 Lost Advance Position... Check Ixxx.x French'
  433 = 'S3 433 Row 44 Lost Return Position... Check Ixxx.x Default' | German: 'S3 433 Row 44 Lost Return Position... Check Ixxx.x German' | French: 'S3 433 Row 44 Lost Return Position... Check Ixxx.x French'
  434 = 'S3 434 Row 44 Switch Fault... Check Ixxx.x / Ixxx.x Default' | German: 'S3 434 Row 44 Switch Fault... Check Ixxx.x / Ixxx.x German' | French: 'S3 434 Row 44 Switch Fault... Check Ixxx.x / Ixxx.x French'
  435 = 'S3 435 Row 44 Spare Message Default' | German: 'S3 435 Row 44 Spare Message German' | French: 'S3 435 Row 44 Spare Message French'
  436 = 'S3 436 Row 44 Spare Message Default' | German: 'S3 436 Row 44 Spare Message German' | French: 'S3 436 Row 44 Spare Message French'
  437 = 'S3 437 Row 44 Spare Message Default' | German: 'S3 437 Row 44 Spare Message German' | French: 'S3 437 Row 44 Spare Message French'
  438 = 'S3 438 Row 44 Spare Message Default' | German: 'S3 438 Row 44 Spare Message German' | French: 'S3 438 Row 44 Spare Message French'
  439 = 'S3 439 Row 44 Spare Message Default' | German: 'S3 439 Row 44 Spare Message German' | French: 'S3 439 Row 44 Spare Message French'
  440 = 'S3 440 Row 45 Failed To Advance.. Check Qxxx.x Default' | German: 'S3 440 Row 45 Failed To Advance.. Check Qxxx.x German' | French: 'S3 440 Row 45 Failed To Advance.. Check Qxxx.x French'
  441 = 'S3 441 Row 45 Failed To Return.. Check Qxxx.x Default' | German: 'S3 441 Row 45 Failed To Return.. Check Qxxx.x German' | French: 'S3 441 Row 45 Failed To Return.. Check Qxxx.x French'
  442 = 'S3 442 Row 45 Lost Advance Position... Check Ixxx.x Default' | German: 'S3 442 Row 45 Lost Advance Position... Check Ixxx.x German' | French: 'S3 442 Row 45 Lost Advance Position... Check Ixxx.x French'
  443 = 'S3 443 Row 45 Lost Return Position... Check Ixxx.x Default' | German: 'S3 443 Row 45 Lost Return Position... Check Ixxx.x German' | French: 'S3 443 Row 45 Lost Return Position... Check Ixxx.x French'
  444 = 'S3 444 Row 45 Switch Fault... Check Ixxx.x / Ixxx.x Default' | German: 'S3 444 Row 45 Switch Fault... Check Ixxx.x / Ixxx.x German' | French: 'S3 444 Row 45 Switch Fault... Check Ixxx.x / Ixxx.x French'
  445 = 'S3 445 Row 45 Spare Message Default' | German: 'S3 445 Row 45 Spare Message German' | French: 'S3 445 Row 45 Spare Message French'
  446 = 'S3 446 Row 45 Spare Message Default' | German: 'S3 446 Row 45 Spare Message German' | French: 'S3 446 Row 45 Spare Message French'
  447 = 'S3 447 Row 45 Spare Message Default' | German: 'S3 447 Row 45 Spare Message German' | French: 'S3 447 Row 45 Spare Message French'
  448 = 'S3 448 Row 45 Spare Message Default' | German: 'S3 448 Row 45 Spare Message German' | French: 'S3 448 Row 45 Spare Message French'
  449 = 'S3 449 Row 45 Spare Message Default' | German: 'S3 449 Row 45 Spare Message German' | French: 'S3 449 Row 45 Spare Message French'
  450 = 'S3 450 Row 46 Failed To Advance.. Check Qxxx.x Default' | German: 'S3 450 Row 46 Failed To Advance.. Check Qxxx.x German' | French: 'S3 450 Row 46 Failed To Advance.. Check Qxxx.x French'
  451 = 'S3 451 Row 46 Failed To Return.. Check Qxxx.x Default' | German: 'S3 451 Row 46 Failed To Return.. Check Qxxx.x German' | French: 'S3 451 Row 46 Failed To Return.. Check Qxxx.x French'
  452 = 'S3 452 Row 46 Lost Advance Position... Check Ixxx.x Default' | German: 'S3 452 Row 46 Lost Advance Position... Check Ixxx.x German' | French: 'S3 452 Row 46 Lost Advance Position... Check Ixxx.x French'
  453 = 'S3 453 Row 46 Lost Return Position... Check Ixxx.x Default' | German: 'S3 453 Row 46 Lost Return Position... Check Ixxx.x German' | French: 'S3 453 Row 46 Lost Return Position... Check Ixxx.x French'
  454 = 'S3 454 Row 46 Switch Fault... Check Ixxx.x / Ixxx.x Default' | German: 'S3 454 Row 46 Switch Fault... Check Ixxx.x / Ixxx.x German' | French: 'S3 454 Row 46 Switch Fault... Check Ixxx.x / Ixxx.x French'
  455 = 'S3 455 Row 46 Spare Message Default' | German: 'S3 455 Row 46 Spare Message German' | French: 'S3 455 Row 46 Spare Message French'
  456 = 'S3 456 Row 46 Spare Message Default' | German: 'S3 456 Row 46 Spare Message German' | French: 'S3 456 Row 46 Spare Message French'
  457 = 'S3 457 Row 46 Spare Message Default' | German: 'S3 457 Row 46 Spare Message German' | French: 'S3 457 Row 46 Spare Message French'
  458 = 'S3 458 Row 46 Spare Message Default' | German: 'S3 458 Row 46 Spare Message German' | French: 'S3 458 Row 46 Spare Message French'
  459 = 'S3 459 Row 46 Spare Message Default' | German: 'S3 459 Row 46 Spare Message German' | French: 'S3 459 Row 46 Spare Message French'
  460 = 'S3 460 Row 47 Failed To Advance.. Check Qxxx.x Default' | German: 'S3 460 Row 47 Failed To Advance.. Check Qxxx.x German' | French: 'S3 460 Row 47 Failed To Advance.. Check Qxxx.x French'
  461 = 'S3 461 Row 47 Failed To Return.. Check Qxxx.x Default' | German: 'S3 461 Row 47 Failed To Return.. Check Qxxx.x German' | French: 'S3 461 Row 47 Failed To Return.. Check Qxxx.x French'
  462 = 'S3 462 Row 47 Lost Advance Position... Check Ixxx.x Default' | German: 'S3 462 Row 47 Lost Advance Position... Check Ixxx.x German' | French: 'S3 462 Row 47 Lost Advance Position... Check Ixxx.x French'
  463 = 'S3 463 Row 47 Lost Return Position... Check Ixxx.x Default' | German: 'S3 463 Row 47 Lost Return Position... Check Ixxx.x German' | French: 'S3 463 Row 47 Lost Return Position... Check Ixxx.x French'
  464 = 'S3 464 Row 47 Switch Fault... Check Ixxx.x / Ixxx.x Default' | German: 'S3 464 Row 47 Switch Fault... Check Ixxx.x / Ixxx.x German' | French: 'S3 464 Row 47 Switch Fault... Check Ixxx.x / Ixxx.x French'
  465 = 'S3 465 Row 47 Spare Message Default' | German: 'S3 465 Row 47 Spare Message German' | French: 'S3 465 Row 47 Spare Message French'
  466 = 'S3 466 Row 47 Spare Message Default' | German: 'S3 466 Row 47 Spare Message German' | French: 'S3 466 Row 47 Spare Message French'
  467 = 'S3 467 Row 47 Spare Message Default' | German: 'S3 467 Row 47 Spare Message German' | French: 'S3 467 Row 47 Spare Message French'
  468 = 'S3 468 Row 47 Spare Message Default' | German: 'S3 468 Row 47 Spare Message German' | French: 'S3 468 Row 47 Spare Message French'
  469 = 'S3 469 Row 47 Spare Message Default' | German: 'S3 469 Row 47 Spare Message German' | French: 'S3 469 Row 47 Spare Message French'
  470 = 'S3 470 Row 48 Failed To Advance.. Check Qxxx.x Default' | German: 'S3 470 Row 48 Failed To Advance.. Check Qxxx.x German' | French: 'S3 470 Row 48 Failed To Advance.. Check Qxxx.x French'
  471 = 'S3 471 Row 48 Failed To Return.. Check Qxxx.x Default' | German: 'S3 471 Row 48 Failed To Return.. Check Qxxx.x German' | French: 'S3 471 Row 48 Failed To Return.. Check Qxxx.x French'
  472 = 'S3 472 Row 48 Lost Advance Position... Check Ixxx.x Default' | German: 'S3 472 Row 48 Lost Advance Position... Check Ixxx.x German' | French: 'S3 472 Row 48 Lost Advance Position... Check Ixxx.x French'
  473 = 'S3 473 Row 48 Lost Return Position... Check Ixxx.x Default' | German: 'S3 473 Row 48 Lost Return Position... Check Ixxx.x German' | French: 'S3 473 Row 48 Lost Return Position... Check Ixxx.x French'
  474 = 'S3 474 Row 48 Switch Fault... Check Ixxx.x / Ixxx.x Default' | German: 'S3 474 Row 48 Switch Fault... Check Ixxx.x / Ixxx.x German' | French: 'S3 474 Row 48 Switch Fault... Check Ixxx.x / Ixxx.x French'
  475 = 'S3 475 Row 48 Spare Message Default' | German: 'S3 475 Row 48 Spare Message German' | French: 'S3 475 Row 48 Spare Message French'
  476 = 'S3 476 Row 48 Spare Message Default' | German: 'S3 476 Row 48 Spare Message German' | French: 'S3 476 Row 48 Spare Message French'
  477 = 'S3 477 Row 48 Spare Message Default' | German: 'S3 477 Row 48 Spare Message German' | French: 'S3 477 Row 48 Spare Message French'
  478 = 'S3 478 Row 48 Spare Message Default' | German: 'S3 478 Row 48 Spare Message German' | French: 'S3 478 Row 48 Spare Message French'
  479 = 'S3 479 Row 48 Spare Message Default' | German: 'S3 479 Row 48 Spare Message German' | French: 'S3 479 Row 48 Spare Message French'
  480 = 'S3 480 Row 49 Failed To Advance.. Check Qxxx.x Default' | German: 'S3 480 Row 49 Failed To Advance.. Check Qxxx.x German' | French: 'S3 480 Row 49 Failed To Advance.. Check Qxxx.x French'
  481 = 'S3 481 Row 49 Failed To Return.. Check Qxxx.x Default' | German: 'S3 481 Row 49 Failed To Return.. Check Qxxx.x German' | French: 'S3 481 Row 49 Failed To Return.. Check Qxxx.x French'
  482 = 'S3 482 Row 49 Lost Advance Position... Check Ixxx.x Default' | German: 'S3 482 Row 49 Lost Advance Position... Check Ixxx.x German' | French: 'S3 482 Row 49 Lost Advance Position... Check Ixxx.x French'
  483 = 'S3 483 Row 49 Lost Return Position... Check Ixxx.x Default' | German: 'S3 483 Row 49 Lost Return Position... Check Ixxx.x German' | French: 'S3 483 Row 49 Lost Return Position... Check Ixxx.x French'
  484 = 'S3 484 Row 49 Switch Fault... Check Ixxx.x / Ixxx.x Default' | German: 'S3 484 Row 49 Switch Fault... Check Ixxx.x / Ixxx.x German' | French: 'S3 484 Row 49 Switch Fault... Check Ixxx.x / Ixxx.x French'
  485 = 'S3 485 Row 49 Spare Message Default' | German: 'S3 485 Row 49 Spare Message German' | French: 'S3 485 Row 49 Spare Message French'
  486 = 'S3 486 Row 49 Spare Message Default' | German: 'S3 486 Row 49 Spare Message German' | French: 'S3 486 Row 49 Spare Message French'
  487 = 'S3 487 Row 49 Spare Message Default' | German: 'S3 487 Row 49 Spare Message German' | French: 'S3 487 Row 49 Spare Message French'
  488 = 'S3 488 Row 49 Spare Message Default' | German: 'S3 488 Row 49 Spare Message German' | French: 'S3 488 Row 49 Spare Message French'
  489 = 'S3 489 Row 49 Spare Message Default' | German: 'S3 489 Row 49 Spare Message German' | French: 'S3 489 Row 49 Spare Message French'
  490 = 'S3 490 Row 50 Failed To Advance.. Check Qxxx.x Default' | German: 'S3 490 Row 50 Failed To Advance.. Check Qxxx.x German' | French: 'S3 490 Row 50 Failed To Advance.. Check Qxxx.x French'
  491 = 'S3 491 Row 50 Failed To Return.. Check Qxxx.x Default' | German: 'S3 491 Row 50 Failed To Return.. Check Qxxx.x German' | French: 'S3 491 Row 50 Failed To Return.. Check Qxxx.x French'
  492 = 'S3 492 Row 50 Lost Advance Position... Check Ixxx.x Default' | German: 'S3 492 Row 50 Lost Advance Position... Check Ixxx.x German' | French: 'S3 492 Row 50 Lost Advance Position... Check Ixxx.x French'
  493 = 'S3 493 Row 50 Lost Return Position... Check Ixxx.x Default' | German: 'S3 493 Row 50 Lost Return Position... Check Ixxx.x German' | French: 'S3 493 Row 50 Lost Return Position... Check Ixxx.x French'
  494 = 'S3 494 Row 50 Switch Fault... Check Ixxx.x / Ixxx.x Default' | German: 'S3 494 Row 50 Switch Fault... Check Ixxx.x / Ixxx.x German' | French: 'S3 494 Row 50 Switch Fault... Check Ixxx.x / Ixxx.x French'
  495 = 'S3 495 Row 50 Spare Message Default' | German: 'S3 495 Row 50 Spare Message German' | French: 'S3 495 Row 50 Spare Message French'
  496 = 'S3 496 Row 50 Spare Message Default' | German: 'S3 496 Row 50 Spare Message German' | French: 'S3 496 Row 50 Spare Message French'
  497 = 'S3 497 Row 50 Spare Message Default' | German: 'S3 497 Row 50 Spare Message German' | French: 'S3 497 Row 50 Spare Message French'
  498 = 'S3 498 Row 50 Spare Message Default' | German: 'S3 498 Row 50 Spare Message German' | French: 'S3 498 Row 50 Spare Message French'
  499 = 'S3 499 Row 50 Spare Message Default' | German: 'S3 499 Row 50 Spare Message German' | French: 'S3 499 Row 50 Spare Message French'
  500 = 'S3 500 Row 51 Failed To Advance.. Check Qxxx.x Default' | German: 'S3 500 Row 51 Failed To Advance.. Check Qxxx.x German' | French: 'S3 500 Row 51 Failed To Advance.. Check Qxxx.x French'
  501 = 'S3 501 Row 51 Failed To Return.. Check Qxxx.x Default' | German: 'S3 501 Row 51 Failed To Return.. Check Qxxx.x German' | French: 'S3 501 Row 51 Failed To Return.. Check Qxxx.x French'
  502 = 'S3 502 Row 51 Lost Advance Position... Check Ixxx.x Default' | German: 'S3 502 Row 51 Lost Advance Position... Check Ixxx.x German' | French: 'S3 502 Row 51 Lost Advance Position... Check Ixxx.x French'
  503 = 'S3 503 Row 51 Lost Return Position... Check Ixxx.x Default' | German: 'S3 503 Row 51 Lost Return Position... Check Ixxx.x German' | French: 'S3 503 Row 51 Lost Return Position... Check Ixxx.x French'
  504 = 'S3 504 Row 51 Switch Fault... Check Ixxx.x / Ixxx.x Default' | German: 'S3 504 Row 51 Switch Fault... Check Ixxx.x / Ixxx.x German' | French: 'S3 504 Row 51 Switch Fault... Check Ixxx.x / Ixxx.x French'
  505 = 'S3 505 Row 51 Spare Message Default' | German: 'S3 505 Row 51 Spare Message German' | French: 'S3 505 Row 51 Spare Message French'
  506 = 'S3 506 Row 51 Spare Message Default' | German: 'S3 506 Row 51 Spare Message German' | French: 'S3 506 Row 51 Spare Message French'
  507 = 'S3 507 Row 51 Spare Message Default' | German: 'S3 507 Row 51 Spare Message German' | French: 'S3 507 Row 51 Spare Message French'
  508 = 'S3 508 Row 51 Spare Message Default' | German: 'S3 508 Row 51 Spare Message German' | French: 'S3 508 Row 51 Spare Message French'
  509 = 'S3 509 Row 51 Spare Message Default' | German: 'S3 509 Row 51 Spare Message German' | French: 'S3 509 Row 51 Spare Message French'
  510 = 'S3 510 Row 52 Failed To Advance.. Check Qxxx.x Default' | German: 'S3 510 Row 52 Failed To Advance.. Check Qxxx.x German' | French: 'S3 510 Row 52 Failed To Advance.. Check Qxxx.x French'
  511 = 'S3 511 Row 52 Failed To Return.. Check Qxxx.x Default' | German: 'S3 511 Row 52 Failed To Return.. Check Qxxx.x German' | French: 'S3 511 Row 52 Failed To Return.. Check Qxxx.x French'
  512 = 'S3 512 Row 52 Lost Advance Position... Check Ixxx.x Default' | German: 'S3 512 Row 52 Lost Advance Position... Check Ixxx.x German' | French: 'S3 512 Row 52 Lost Advance Position... Check Ixxx.x French'
  513 = 'S3 513 Row 52 Lost Return Position... Check Ixxx.x Default' | German: 'S3 513 Row 52 Lost Return Position... Check Ixxx.x German' | French: 'S3 513 Row 52 Lost Return Position... Check Ixxx.x French'
  514 = 'S3 514 Row 52 Switch Fault... Check Ixxx.x / Ixxx.x Default' | German: 'S3 514 Row 52 Switch Fault... Check Ixxx.x / Ixxx.x German' | French: 'S3 514 Row 52 Switch Fault... Check Ixxx.x / Ixxx.x French'
  515 = 'S3 515 Row 52 Spare Message Default' | German: 'S3 515 Row 52 Spare Message German' | French: 'S3 515 Row 52 Spare Message French'
  516 = 'S3 516 Row 52 Spare Message Default' | German: 'S3 516 Row 52 Spare Message German' | French: 'S3 516 Row 52 Spare Message French'
  517 = 'S3 517 Row 52 Spare Message Default' | German: 'S3 517 Row 52 Spare Message German' | French: 'S3 517 Row 52 Spare Message French'
  518 = 'S3 518 Row 52 Spare Message Default' | German: 'S3 518 Row 52 Spare Message German' | French: 'S3 518 Row 52 Spare Message French'
  519 = 'S3 519 Row 52 Spare Message Default' | German: 'S3 519 Row 52 Spare Message German' | French: 'S3 519 Row 52 Spare Message French'
  520 = 'S3 520 Row 53 Failed To Advance.. Check Qxxx.x Default' | German: 'S3 520 Row 53 Failed To Advance.. Check Qxxx.x German' | French: 'S3 520 Row 53 Failed To Advance.. Check Qxxx.x French'
  521 = 'S3 521 Row 53 Failed To Return.. Check Qxxx.x Default' | German: 'S3 521 Row 53 Failed To Return.. Check Qxxx.x German' | French: 'S3 521 Row 53 Failed To Return.. Check Qxxx.x French'
  522 = 'S3 522 Row 53 Lost Advance Position... Check Ixxx.x Default' | German: 'S3 522 Row 53 Lost Advance Position... Check Ixxx.x German' | French: 'S3 522 Row 53 Lost Advance Position... Check Ixxx.x French'
  523 = 'S3 523 Row 53 Lost Return Position... Check Ixxx.x Default' | German: 'S3 523 Row 53 Lost Return Position... Check Ixxx.x German' | French: 'S3 523 Row 53 Lost Return Position... Check Ixxx.x French'
  524 = 'S3 524 Row 53 Switch Fault... Check Ixxx.x / Ixxx.x Default' | German: 'S3 524 Row 53 Switch Fault... Check Ixxx.x / Ixxx.x German' | French: 'S3 524 Row 53 Switch Fault... Check Ixxx.x / Ixxx.x French'
  525 = 'S3 525 Row 53 Spare Message Default' | German: 'S3 525 Row 53 Spare Message German' | French: 'S3 525 Row 53 Spare Message French'
  526 = 'S3 526 Row 53 Spare Message Default' | German: 'S3 526 Row 53 Spare Message German' | French: 'S3 526 Row 53 Spare Message French'
  527 = 'S3 527 Row 53 Spare Message Default' | German: 'S3 527 Row 53 Spare Message German' | French: 'S3 527 Row 53 Spare Message French'
  528 = 'S3 528 Row 53 Spare Message Default' | German: 'S3 528 Row 53 Spare Message German' | French: 'S3 528 Row 53 Spare Message French'
  529 = 'S3 529 Row 53 Spare Message Default' | German: 'S3 529 Row 53 Spare Message German' | French: 'S3 529 Row 53 Spare Message French'
  530 = 'S3 530 Row 54 Failed To Advance.. Check Qxxx.x Default' | German: 'S3 530 Row 54 Failed To Advance.. Check Qxxx.x German' | French: 'S3 530 Row 54 Failed To Advance.. Check Qxxx.x French'
  531 = 'S3 531 Row 54 Failed To Return.. Check Qxxx.x Default' | German: 'S3 531 Row 54 Failed To Return.. Check Qxxx.x German' | French: 'S3 531 Row 54 Failed To Return.. Check Qxxx.x French'
  532 = 'S3 532 Row 54 Lost Advance Position... Check Ixxx.x Default' | German: 'S3 532 Row 54 Lost Advance Position... Check Ixxx.x German' | French: 'S3 532 Row 54 Lost Advance Position... Check Ixxx.x French'
  533 = 'S3 533 Row 54 Lost Return Position... Check Ixxx.x Default' | German: 'S3 533 Row 54 Lost Return Position... Check Ixxx.x German' | French: 'S3 533 Row 54 Lost Return Position... Check Ixxx.x French'
  534 = 'S3 534 Row 54 Switch Fault... Check Ixxx.x / Ixxx.x Default' | German: 'S3 534 Row 54 Switch Fault... Check Ixxx.x / Ixxx.x German' | French: 'S3 534 Row 54 Switch Fault... Check Ixxx.x / Ixxx.x French'
  535 = 'S3 535 Row 54 Spare Message Default' | German: 'S3 535 Row 54 Spare Message German' | French: 'S3 535 Row 54 Spare Message French'
  536 = 'S3 536 Row 54 Spare Message Default' | German: 'S3 536 Row 54 Spare Message German' | French: 'S3 536 Row 54 Spare Message French'
  537 = 'S3 537 Row 54 Spare Message Default' | German: 'S3 537 Row 54 Spare Message German' | French: 'S3 537 Row 54 Spare Message French'
  538 = 'S3 538 Row 54 Spare Message Default' | German: 'S3 538 Row 54 Spare Message German' | French: 'S3 538 Row 54 Spare Message French'
  539 = 'S3 539 Row 54 Spare Message Default' | German: 'S3 539 Row 54 Spare Message German' | French: 'S3 539 Row 54 Spare Message French'
  540 = 'S3 540 Row 55 Failed To Advance.. Check Qxxx.x Default' | German: 'S3 540 Row 55 Failed To Advance.. Check Qxxx.x German' | French: 'S3 540 Row 55 Failed To Advance.. Check Qxxx.x French'
  541 = 'S3 541 Row 55 Failed To Return.. Check Qxxx.x Default' | German: 'S3 541 Row 55 Failed To Return.. Check Qxxx.x German' | French: 'S3 541 Row 55 Failed To Return.. Check Qxxx.x French'
  542 = 'S3 542 Row 55 Lost Advance Position... Check Ixxx.x Default' | German: 'S3 542 Row 55 Lost Advance Position... Check Ixxx.x German' | French: 'S3 542 Row 55 Lost Advance Position... Check Ixxx.x French'
  543 = 'S3 543 Row 55 Lost Return Position... Check Ixxx.x Default' | German: 'S3 543 Row 55 Lost Return Position... Check Ixxx.x German' | French: 'S3 543 Row 55 Lost Return Position... Check Ixxx.x French'
  544 = 'S3 544 Row 55 Switch Fault... Check Ixxx.x / Ixxx.x Default' | German: 'S3 544 Row 55 Switch Fault... Check Ixxx.x / Ixxx.x German' | French: 'S3 544 Row 55 Switch Fault... Check Ixxx.x / Ixxx.x French'
  545 = 'S3 545 Row 55 Spare Message Default' | German: 'S3 545 Row 55 Spare Message German' | French: 'S3 545 Row 55 Spare Message French'
  546 = 'S3 546 Row 55 Spare Message Default' | German: 'S3 546 Row 55 Spare Message German' | French: 'S3 546 Row 55 Spare Message French'
  547 = 'S3 547 Row 55 Spare Message Default' | German: 'S3 547 Row 55 Spare Message German' | French: 'S3 547 Row 55 Spare Message French'
  548 = 'S3 548 Row 55 Spare Message Default' | German: 'S3 548 Row 55 Spare Message German' | French: 'S3 548 Row 55 Spare Message French'
  549 = 'S3 549 Row 55 Spare Message Default' | German: 'S3 549 Row 55 Spare Message German' | French: 'S3 549 Row 55 Spare Message French'
  550 = 'S3 550 Row 56 Failed To Advance.. Check Qxxx.x Default' | German: 'S3 550 Row 56 Failed To Advance.. Check Qxxx.x German' | French: 'S3 550 Row 56 Failed To Advance.. Check Qxxx.x French'
  551 = 'S3 551 Row 56 Failed To Return.. Check Qxxx.x Default' | German: 'S3 551 Row 56 Failed To Return.. Check Qxxx.x German' | French: 'S3 551 Row 56 Failed To Return.. Check Qxxx.x French'
  552 = 'S3 552 Row 56 Lost Advance Position... Check Ixxx.x Default' | German: 'S3 552 Row 56 Lost Advance Position... Check Ixxx.x German' | French: 'S3 552 Row 56 Lost Advance Position... Check Ixxx.x French'
  553 = 'S3 553 Row 56 Lost Return Position... Check Ixxx.x Default' | German: 'S3 553 Row 56 Lost Return Position... Check Ixxx.x German' | French: 'S3 553 Row 56 Lost Return Position... Check Ixxx.x French'
  554 = 'S3 554 Row 56 Switch Fault... Check Ixxx.x / Ixxx.x Default' | German: 'S3 554 Row 56 Switch Fault... Check Ixxx.x / Ixxx.x German' | French: 'S3 554 Row 56 Switch Fault... Check Ixxx.x / Ixxx.x French'
  555 = 'S3 555 Row 56 Spare Message Default' | German: 'S3 555 Row 56 Spare Message German' | French: 'S3 555 Row 56 Spare Message French'
  556 = 'S3 556 Row 56 Spare Message Default' | German: 'S3 556 Row 56 Spare Message German' | French: 'S3 556 Row 56 Spare Message French'
  557 = 'S3 557 Row 56 Spare Message Default' | German: 'S3 557 Row 56 Spare Message German' | French: 'S3 557 Row 56 Spare Message French'
  558 = 'S3 558 Row 56 Spare Message Default' | German: 'S3 558 Row 56 Spare Message German' | French: 'S3 558 Row 56 Spare Message French'
  559 = 'S3 559 Row 56 Spare Message Default' | German: 'S3 559 Row 56 Spare Message German' | French: 'S3 559 Row 56 Spare Message French'
  560 = 'S3 560 Row 57 Failed To Advance.. Check Qxxx.x Default' | German: 'S3 560 Row 57 Failed To Advance.. Check Qxxx.x German' | French: 'S3 560 Row 57 Failed To Advance.. Check Qxxx.x French'
  561 = 'S3 561 Row 57 Failed To Return.. Check Qxxx.x Default' | German: 'S3 561 Row 57 Failed To Return.. Check Qxxx.x German' | French: 'S3 561 Row 57 Failed To Return.. Check Qxxx.x French'
  562 = 'S3 562 Row 57 Lost Advance Position... Check Ixxx.x Default' | German: 'S3 562 Row 57 Lost Advance Position... Check Ixxx.x German' | French: 'S3 562 Row 57 Lost Advance Position... Check Ixxx.x French'
  563 = 'S3 563 Row 57 Lost Return Position... Check Ixxx.x Default' | German: 'S3 563 Row 57 Lost Return Position... Check Ixxx.x German' | French: 'S3 563 Row 57 Lost Return Position... Check Ixxx.x French'
  564 = 'S3 564 Row 57 Switch Fault... Check Ixxx.x / Ixxx.x Default' | German: 'S3 564 Row 57 Switch Fault... Check Ixxx.x / Ixxx.x German' | French: 'S3 564 Row 57 Switch Fault... Check Ixxx.x / Ixxx.x French'
  565 = 'S3 565 Row 57 Spare Message Default' | German: 'S3 565 Row 57 Spare Message German' | French: 'S3 565 Row 57 Spare Message French'
  566 = 'S3 566 Row 57 Spare Message Default' | German: 'S3 566 Row 57 Spare Message German' | French: 'S3 566 Row 57 Spare Message French'
  567 = 'S3 567 Row 57 Spare Message Default' | German: 'S3 567 Row 57 Spare Message German' | French: 'S3 567 Row 57 Spare Message French'
  568 = 'S3 568 Row 57 Spare Message Default' | German: 'S3 568 Row 57 Spare Message German' | French: 'S3 568 Row 57 Spare Message French'
  569 = 'S3 569 Row 57 Spare Message Default' | German: 'S3 569 Row 57 Spare Message German' | French: 'S3 569 Row 57 Spare Message French'
  570 = 'S3 570 Row 58 Failed To Advance.. Check Qxxx.x Default' | German: 'S3 570 Row 58 Failed To Advance.. Check Qxxx.x German' | French: 'S3 570 Row 58 Failed To Advance.. Check Qxxx.x French'
  571 = 'S3 571 Row 58 Failed To Return.. Check Qxxx.x Default' | German: 'S3 571 Row 58 Failed To Return.. Check Qxxx.x German' | French: 'S3 571 Row 58 Failed To Return.. Check Qxxx.x French'
  572 = 'S3 572 Row 58 Lost Advance Position... Check Ixxx.x Default' | German: 'S3 572 Row 58 Lost Advance Position... Check Ixxx.x German' | French: 'S3 572 Row 58 Lost Advance Position... Check Ixxx.x French'
  573 = 'S3 573 Row 58 Lost Return Position... Check Ixxx.x Default' | German: 'S3 573 Row 58 Lost Return Position... Check Ixxx.x German' | French: 'S3 573 Row 58 Lost Return Position... Check Ixxx.x French'
  574 = 'S3 574 Row 58 Switch Fault... Check Ixxx.x / Ixxx.x Default' | German: 'S3 574 Row 58 Switch Fault... Check Ixxx.x / Ixxx.x German' | French: 'S3 574 Row 58 Switch Fault... Check Ixxx.x / Ixxx.x French'
  575 = 'S3 575 Row 58 Spare Message Default' | German: 'S3 575 Row 58 Spare Message German' | French: 'S3 575 Row 58 Spare Message French'
  576 = 'S3 576 Row 58 Spare Message Default' | German: 'S3 576 Row 58 Spare Message German' | French: 'S3 576 Row 58 Spare Message French'
  577 = 'S3 577 Row 58 Spare Message Default' | German: 'S3 577 Row 58 Spare Message German' | French: 'S3 577 Row 58 Spare Message French'
  578 = 'S3 578 Row 58 Spare Message Default' | German: 'S3 578 Row 58 Spare Message German' | French: 'S3 578 Row 58 Spare Message French'
  579 = 'S3 579 Row 58 Spare Message Default' | German: 'S3 579 Row 58 Spare Message German' | French: 'S3 579 Row 58 Spare Message French'
  580 = 'S3 580 Row 59 Failed To Advance.. Check Qxxx.x Default' | German: 'S3 580 Row 59 Failed To Advance.. Check Qxxx.x German' | French: 'S3 580 Row 59 Failed To Advance.. Check Qxxx.x French'
  581 = 'S3 581 Row 59 Failed To Return.. Check Qxxx.x Default' | German: 'S3 581 Row 59 Failed To Return.. Check Qxxx.x German' | French: 'S3 581 Row 59 Failed To Return.. Check Qxxx.x French'
  582 = 'S3 582 Row 59 Lost Advance Position... Check Ixxx.x Default' | German: 'S3 582 Row 59 Lost Advance Position... Check Ixxx.x German' | French: 'S3 582 Row 59 Lost Advance Position... Check Ixxx.x French'
